C01823=1131.595,336.881,-80.038,-177.462,10.810,149.511
C01824=1131.592,337.129,-80.073,-177.459,10.813,149.510
C01825=1131.587,337.377,-80.107,-177.456,10.816,149.510
C01826=1131.583,337.624,-80.141,-177.452,10.818,149.510
C01827=1131.579,337.872,-80.176,-177.449,10.821,149.510
C01828=1131.576,338.119,-80.210,-177.446,10.823,149.510
C01829=1131.572,338.367,-80.244,-177.442,10.826,149.509
C01830=1131.568,338.614,-80.278,-177.439,10.828,149.509
C01831=1131.564,338.862,-80.313,-177.436,10.831,149.509
C01832=1131.560,339.109,-80.347,-177.433,10.833,149.509
C01833=1131.556,339.357,-80.382,-177.429,10.836,149.509
C01834=1131.552,339.605,-80.416,-177.426,10.838,149.508
C01835=1131.548,339.852,-80.450,-177.423,10.841,149.508
C01836=1131.544,340.100,-80.485,-177.421,10.843,149.508
C01837=1131.540,340.347,-80.519,-177.417,10.845,149.508
C01838=1131.536,340.595,-80.554,-177.414,10.847,149.508
C01839=1131.532,340.842,-80.588,-177.411,10.850,149.507
C01840=1131.528,341.091,-80.622,-177.407,10.852,149.507
C01841=1131.524,341.338,-80.657,-177.404,10.855,149.507
C01842=1131.520,341.586,-80.691,-177.401,10.858,149.507
C01843=1131.516,341.833,-80.726,-177.398,10.860,149.507
C01844=1131.512,342.081,-80.760,-177.394,10.863,149.506
C01845=1131.508,342.328,-80.795,-177.391,10.865,149.506
C01846=1131.504,342.576,-80.830,-177.388,10.867,149.506
C01847=1131.500,342.823,-80.864,-177.385,10.870,149.506
C01848=1131.496,343.071,-80.898,-177.382,10.873,149.506
C01849=1131.492,343.319,-80.933,-177.378,10.875,149.505
C01850=1131.488,343.566,-80.969,-177.375,10.878,149.505
C01851=1131.484,343.813,-81.002,-177.372,10.880,149.505
C01852=1131.480,344.061,-81.037,-177.368,10.883,149.505
C01853=1131.476,344.309,-81.072,-177.365,10.885,149.505
C01854=1131.473,344.556,-81.107,-177.362,10.888,149.504
C01855=1131.469,344.804,-81.141,-177.359,10.890,149.504
C01856=1131.464,345.051,-81.176,-177.355,10.893,149.504
C01857=1131.461,345.299,-81.211,-177.352,10.895,149.504
C01858=1131.457,345.546,-81.245,-177.349,10.898,149.503
C01859=1131.453,345.794,-81.280,-177.345,10.900,149.503
C01860=1131.449,346.042,-81.316,-177.343,10.903,149.503
C01861=1131.445,346.289,-81.350,-177.339,10.905,149.503
C01862=1131.441,346.537,-81.386,-177.336,10.908,149.503
C01863=1131.437,346.784,-81.420,-177.333,10.910,149.502
C01864=1131.433,347.032,-81.454,-177.329,10.913,149.502
C01865=1131.430,347.279,-81.490,-177.326,10.915,149.502
C01866=1131.425,347.527,-81.524,-177.323,10.918,149.502
C01867=1131.421,347.774,-81.560,-177.319,10.920,149.502
C01868=1131.419,347.987,-81.590,-177.317,10.922,149.501
C01869=1131.414,348.200,-81.619,-177.314,10.924,149.501
C01870=1131.411,348.414,-81.650,-177.311,10.927,149.501
C01871=1131.408,348.626,-81.680,-177.309,10.928,149.501
C01872=1131.405,348.839,-81.710,-177.305,10.931,149.501
C01873=1131.401,349.052,-81.741,-177.303,10.933,149.501
C01874=1131.398,349.265,-81.770,-177.300,10.935,149.500
C01875=1131.395,349.478,-81.801,-177.297,10.937,149.500
C01876=1131.391,349.726,-81.836,-177.294,10.939,149.500
C01877=1131.386,349.973,-81.871,-177.290,10.943,149.500
C01878=1131.383,350.220,-81.906,-177.287,10.945,149.499
C01879=1131.379,350.469,-81.941,-177.282,10.948,149.499
C01880=1131.375,350.716,-81.977,-177.279,10.950,149.499
C01881=1131.371,350.963,-82.012,-177.275,10.954,149.499
C01882=1131.367,351.211,-82.047,-177.272,10.956,149.498
C01883=1131.363,351.459,-82.082,-177.268,10.958,149.498
C01884=1131.359,351.705,-82.118,-177.264,10.961,149.498
C01885=1131.355,351.953,-82.152,-177.261,10.964,149.498
C01886=1131.351,352.201,-82.188,-177.257,10.966,149.497
C01887=1131.348,352.448,-82.224,-177.253,10.969,149.497
C01888=1131.343,352.695,-82.259,-177.250,10.972,149.497
C01889=1131.340,352.943,-82.294,-177.247,10.974,149.497
C01890=1131.336,353.191,-82.329,-177.242,10.977,149.496
C01891=1131.332,353.438,-82.365,-177.239,10.980,149.496
C01892=1131.328,353.686,-82.400,-177.236,10.982,149.496
C01893=1131.324,353.933,-82.435,-177.231,10.985,149.495
C01894=1131.321,354.180,-82.471,-177.228,10.987,149.495
C01895=1131.317,354.428,-82.506,-177.225,10.990,149.495
C01896=1131.313,354.675,-82.542,-177.221,10.992,149.495
C01897=1131.310,354.923,-82.578,-177.217,10.995,149.494
C01898=1131.305,355.169,-82.613,-177.214,10.998,149.494
C01899=1131.302,355.417,-82.648,-177.210,11.000,149.494
C01900=1131.297,355.665,-82.684,-177.207,11.002,149.493
C01901=1131.294,355.912,-82.720,-177.203,11.006,149.493
C01902=1131.290,356.160,-82.756,-177.199,11.008,149.493
C01903=1131.286,356.407,-82.791,-177.196,11.010,149.493
C01904=1131.282,356.654,-82.826,-177.192,11.013,149.492
C01905=1131.278,356.902,-82.862,-177.189,11.015,149.492
C01906=1131.274,357.149,-82.898,-177.185,11.018,149.492
C01907=1131.270,357.397,-82.933,-177.181,11.020,149.492
C01908=1131.267,357.644,-82.969,-177.178,11.023,149.491
C01909=1131.263,357.892,-83.005,-177.175,11.025,149.491
C01910=1131.259,358.139,-83.040,-177.171,11.028,149.491
C01911=1131.255,358.387,-83.077,-177.168,11.030,149.491
C01912=1131.251,358.633,-83.112,-177.164,11.032,149.490
C01913=1131.247,358.881,-83.148,-177.161,11.035,149.490
C01914=1131.244,359.128,-83.183,-177.158,11.037,149.490
C01915=1131.239,359.376,-83.219,-177.154,11.040,149.490
C01916=1131.236,359.623,-83.256,-177.150,11.043,149.489
C01917=1131.232,359.871,-83.291,-177.147,11.045,149.489
C01918=1131.228,360.118,-83.327,-177.143,11.047,149.489
C01919=1131.224,360.366,-83.363,-177.140,11.050,149.488
C01920=1131.221,360.613,-83.399,-177.137,11.052,149.488
C01921=1131.217,360.860,-83.435,-177.133,11.055,149.488
C01922=1131.213,361.108,-83.471,-177.130,11.057,149.488
C01923=1131.209,361.355,-83.507,-177.126,11.059,149.487
C01924=1131.206,361.568,-83.538,-177.124,11.061,149.487
C01925=1131.203,361.781,-83.569,-177.120,11.064,149.487
C01926=1131.199,361.993,-83.600,-177.118,11.066,149.487
C01927=1131.196,362.206,-83.630,-177.115,11.068,149.487
C01928=1131.193,362.419,-83.662,-177.112,11.070,149.486
C01929=1131.190,362.631,-83.693,-177.109,11.071,149.486
C01930=1131.186,362.845,-83.724,-177.106,11.074,149.486
C01931=1131.183,363.058,-83.755,-177.103,11.076,149.486
C01932=1131.179,363.305,-83.791,-177.100,11.078,149.485
C01933=1131.176,363.552,-83.827,-177.097,11.080,149.485
C01934=1131.171,363.800,-83.863,-177.093,11.083,149.485
C01935=1131.168,364.047,-83.900,-177.090,11.085,149.485
C01936=1131.163,364.295,-83.936,-177.086,11.088,149.484
C01937=1131.160,364.541,-83.972,-177.083,11.090,149.484
C01938=1131.156,364.789,-84.008,-177.080,11.093,149.484
C01939=1131.152,365.036,-84.044,-177.077,11.095,149.484
C01940=1131.148,365.283,-84.081,-177.074,11.097,149.484
C01941=1131.145,365.531,-84.117,-177.070,11.099,149.483
C01942=1131.141,365.778,-84.154,-177.067,11.101,149.483
C01943=1131.137,366.025,-84.189,-177.064,11.104,149.483
C01944=1131.133,366.273,-84.226,-177.060,11.106,149.483
C01945=1131.130,366.520,-84.263,-177.057,11.109,149.482
C01946=1131.126,366.768,-84.299,-177.054,11.111,149.482
C01947=1131.122,367.015,-84.335,-177.051,11.113,149.482
C01948=1131.118,367.262,-84.372,-177.048,11.115,149.482
C01949=1131.115,367.510,-84.408,-177.044,11.118,149.481
C01950=1131.110,367.757,-84.444,-177.041,11.120,149.481
C01951=1131.106,368.004,-84.481,-177.038,11.123,149.481
C01952=1131.103,368.251,-84.518,-177.035,11.124,149.481
C01953=1131.099,368.499,-84.554,-177.032,11.127,149.481
C01954=1131.095,368.746,-84.590,-177.029,11.129,149.480
C01955=1131.092,368.993,-84.627,-177.025,11.132,149.480
C01956=1131.088,369.241,-84.664,-177.023,11.134,149.480
C01957=1131.084,369.488,-84.700,-177.019,11.136,149.480
C01958=1131.080,369.735,-84.736,-177.016,11.139,149.479
C01959=1131.076,369.982,-84.773,-177.013,11.141,149.479
C01960=1131.072,370.229,-84.810,-177.010,11.143,149.479
C01961=1131.068,370.477,-84.846,-177.007,11.145,149.479
C01962=1131.066,370.724,-84.883,-177.003,11.148,149.479
C01963=1131.061,370.971,-84.920,-177.000,11.150,149.478
C01964=1131.057,371.219,-84.957,-176.997,11.152,149.478
C01965=1131.053,371.466,-84.994,-176.994,11.154,149.478
C01966=1131.050,371.713,-85.030,-176.991,11.157,149.478
C01967=1131.046,371.961,-85.066,-176.989,11.159,149.478
C01968=1131.042,372.208,-85.103,-176.985,11.161,149.477
C01969=1131.039,372.455,-85.139,-176.982,11.164,149.477
C01970=1131.035,372.702,-85.176,-176.979,11.166,149.477
C01971=1131.030,372.950,-85.213,-176.976,11.168,149.477
C01972=1131.027,373.198,-85.250,-176.973,11.170,149.477
C01973=1131.024,373.444,-85.287,-176.970,11.173,149.477
C01974=1131.020,373.691,-85.324,-176.967,11.175,149.476
C01975=1131.016,373.938,-85.361,-176.964,11.177,149.476
C01976=1131.012,374.185,-85.398,-176.961,11.179,149.476
C01977=1131.009,374.433,-85.435,-176.958,11.182,149.476
C01978=1131.005,374.680,-85.471,-176.955,11.184,149.476
C01979=1131.001,374.927,-85.508,-176.952,11.186,149.475
C01980=1130.997,375.140,-85.540,-176.950,11.188,149.475
C01981=1130.994,375.352,-85.572,-176.947,11.191,149.475
C01982=1130.991,375.565,-85.603,-176.944,11.193,149.475
C01983=1130.988,375.779,-85.636,-176.942,11.195,149.475
C01984=1130.985,375.991,-85.668,-176.939,11.196,149.475
C01985=1130.981,376.204,-85.700,-176.937,11.198,149.475
C01986=1130.978,376.416,-85.731,-176.935,11.200,149.474
C01987=1130.975,376.629,-85.763,-176.932,11.202,149.474
C01988=1130.971,376.876,-85.800,-176.929,11.205,149.474
C01989=1130.967,377.124,-85.838,-176.927,11.207,149.474
C01990=1130.963,377.371,-85.874,-176.923,11.209,149.474
C01991=1130.960,377.618,-85.911,-176.921,11.211,149.474
C01992=1130.956,377.864,-85.948,-176.918,11.214,149.474
C01993=1130.953,378.112,-85.985,-176.915,11.216,149.474
C01994=1130.948,378.359,-86.022,-176.912,11.218,149.473
C01995=1130.945,378.606,-86.060,-176.909,11.221,149.473
C01996=1130.941,378.854,-86.097,-176.907,11.223,149.473
C01997=1130.937,379.101,-86.134,-176.904,11.225,149.473
C01998=1130.933,379.348,-86.172,-176.901,11.227,149.473
C01999=1130.930,379.596,-86.209,-176.898,11.230,149.473
C02000=1130.926,379.843,-86.246,-176.896,11.232,149.473
C02001=1130.922,380.089,-86.283,-176.893,11.235,149.473
C02002=1130.918,380.337,-86.320,-176.890,11.236,149.473
C02003=1130.915,380.584,-86.358,-176.887,11.239,149.473
C02004=1130.911,380.831,-86.395,-176.885,11.241,149.473
C02005=1130.907,381.078,-86.433,-176.882,11.244,149.472
C02006=1130.903,381.325,-86.470,-176.880,11.246,149.472
C02007=1130.899,381.573,-86.506,-176.877,11.249,149.472
C02008=1130.896,381.820,-86.544,-176.874,11.251,149.472
C02009=1130.892,382.067,-86.581,-176.871,11.253,149.472
C02010=1130.889,382.314,-86.619,-176.869,11.255,149.472
C02011=1130.885,382.562,-86.656,-176.866,11.258,149.472
C02012=1130.881,382.808,-86.694,-176.864,11.260,149.472
C02013=1130.878,383.055,-86.732,-176.861,11.263,149.472
C02014=1130.874,383.303,-86.768,-176.859,11.265,149.472
C02015=1130.870,383.550,-86.806,-176.856,11.267,149.472
C02016=1130.866,383.797,-86.843,-176.855,11.268,149.472
C02017=1130.862,384.044,-86.881,-176.854,11.270,149.472
C02018=1130.858,384.292,-86.919,-176.853,11.272,149.472
C02019=1130.854,384.538,-86.956,-176.852,11.273,149.472
C02020=1130.851,384.786,-86.994,-176.850,11.275,149.472
C02021=1130.847,385.033,-87.031,-176.849,11.277,149.473
C02022=1130.844,385.280,-87.069,-176.847,11.279,149.473
C02023=1130.840,385.527,-87.106,-176.846,11.281,149.473
C02024=1130.836,385.774,-87.143,-176.845,11.282,149.473
C02025=1130.833,386.021,-87.181,-176.844,11.284,149.473
C02026=1130.829,386.268,-87.218,-176.843,11.286,149.473
C02027=1130.825,386.516,-87.257,-176.842,11.288,149.473
C02028=1130.821,386.762,-87.294,-176.841,11.289,149.474
C02029=1130.818,387.010,-87.332,-176.840,11.291,149.474
C02030=1130.814,387.257,-87.369,-176.838,11.293,149.474
C02031=1130.811,387.504,-87.407,-176.837,11.295,149.474
C02032=1130.807,387.751,-87.444,-176.836,11.297,149.474
C02033=1130.803,387.999,-87.482,-176.835,11.299,149.475
C02034=1130.799,388.246,-87.520,-176.834,11.301,149.475
C02035=1130.795,388.492,-87.558,-176.833,11.303,149.475
C02036=1130.793,388.705,-87.589,-176.832,11.304,149.475
C02037=1130.789,388.918,-87.622,-176.831,11.306,149.475
C02038=1130.786,389.130,-87.654,-176.830,11.308,149.476
C02039=1130.782,389.342,-87.687,-176.830,11.309,149.476
C02040=1130.780,389.555,-87.719,-176.829,11.311,149.476
C02041=1130.776,389.768,-87.751,-176.828,11.313,149.477
C02042=1130.773,389.981,-87.784,-176.827,11.315,149.477
C02043=1130.769,390.193,-87.816,-176.827,11.317,149.477
C02044=1130.766,390.440,-87.854,-176.826,11.319,149.477
C02045=1130.762,390.687,-87.892,-176.825,11.320,149.478
C02046=1130.759,390.935,-87.929,-176.824,11.322,149.478
C02047=1130.755,391.181,-87.967,-176.824,11.325,149.478
C02048=1130.751,391.429,-88.005,-176.822,11.327,149.479
C02049=1130.747,391.675,-88.043,-176.822,11.329,149.479
C02050=1130.744,391.923,-88.080,-176.821,11.331,149.479
C02051=1130.740,392.170,-88.118,-176.820,11.334,149.480
C02052=1130.737,392.417,-88.156,-176.819,11.335,149.480
C02053=1130.732,392.664,-88.194,-176.818,11.339,149.481
C02054=1130.729,392.911,-88.232,-176.817,11.340,149.481
C02055=1130.725,393.158,-88.269,-176.817,11.343,149.481
C02056=1130.722,393.406,-88.306,-176.817,11.345,149.482
C02057=1130.717,393.653,-88.345,-176.816,11.347,149.482
C02058=1130.714,393.900,-88.383,-176.815,11.350,149.483
C02059=1130.710,394.146,-88.420,-176.815,11.352,149.483
C02060=1130.707,394.394,-88.458,-176.814,11.355,149.484
C02061=1130.703,394.641,-88.496,-176.814,11.357,149.484
C02062=1130.699,394.888,-88.534,-176.813,11.359,149.485
C02063=1130.696,395.136,-88.571,-176.812,11.362,149.485
C02064=1130.692,395.382,-88.609,-176.812,11.364,149.486
C02065=1130.688,395.630,-88.648,-176.811,11.366,149.486
C02066=1130.684,395.876,-88.685,-176.811,11.369,149.487
C02067=1130.681,396.124,-88.723,-176.810,11.372,149.487
C02068=1130.677,396.371,-88.761,-176.810,11.374,149.488
C02069=1130.674,396.618,-88.799,-176.809,11.377,149.488
C02070=1130.670,396.864,-88.837,-176.809,11.379,149.489
C02071=1130.667,397.112,-88.875,-176.808,11.382,149.490
C02072=1130.662,397.359,-88.913,-176.808,11.385,149.490
C02073=1130.659,397.606,-88.951,-176.808,11.387,149.491
C02074=1130.655,397.853,-88.988,-176.807,11.391,149.491
C02075=1130.651,398.101,-89.026,-176.807,11.393,149.492
C02076=1130.647,398.347,-89.064,-176.807,11.396,149.493
C02077=1130.644,398.594,-89.102,-176.807,11.398,149.493
C02078=1130.640,398.842,-89.140,-176.806,11.402,149.494
C02079=1130.636,399.089,-89.178,-176.806,11.404,149.495
C02080=1130.633,399.336,-89.216,-176.806,11.407,149.495
C02081=1130.628,399.583,-89.254,-176.805,11.410,149.496
C02082=1130.625,399.830,-89.292,-176.805,11.413,149.497
C02083=1130.621,400.077,-89.329,-176.805,11.415,149.497
C02084=1130.618,400.324,-89.368,-176.805,11.419,149.498
C02085=1130.614,400.571,-89.406,-176.805,11.421,149.499
C02086=1130.611,400.818,-89.443,-176.804,11.425,149.499
C02087=1130.607,401.066,-89.482,-176.804,11.428,149.500
C02088=1130.603,401.312,-89.520,-176.805,11.430,149.501
C02089=1130.600,401.559,-89.557,-176.804,11.434,149.502
C02090=1130.595,401.806,-89.596,-176.804,11.437,149.503
C02091=1130.592,402.054,-89.634,-176.805,11.440,149.503
C02092=1130.589,402.265,-89.667,-176.804,11.443,149.504
C02093=1130.586,402.478,-89.700,-176.804,11.445,149.505
C02094=1130.582,402.691,-89.732,-176.804,11.448,149.506
C02095=1130.579,402.903,-89.765,-176.804,11.451,149.506
C02096=1130.577,403.116,-89.797,-176.804,11.454,149.507
C02097=1130.573,403.328,-89.830,-176.804,11.456,149.508
C02098=1130.570,403.540,-89.863,-176.805,11.459,149.509
C02099=1130.567,403.754,-89.896,-176.805,11.462,149.509
C02100=1130.562,404.000,-89.934,-176.804,11.465,149.510
C02101=1130.560,404.247,-89.972,-176.805,11.469,149.511
C02102=1130.556,404.494,-90.010,-176.805,11.472,149.512
C02103=1130.552,404.741,-90.048,-176.805,11.476,149.513
C02104=1130.549,404.988,-90.086,-176.805,11.479,149.514
C02105=1130.544,405.235,-90.125,-176.806,11.482,149.515
C02106=1130.541,405.483,-90.162,-176.805,11.486,149.516
C02107=1130.537,405.729,-90.200,-176.806,11.489,149.517
C02108=1130.533,405.977,-90.239,-176.806,11.493,149.518
C02109=1130.530,406.223,-90.277,-176.807,11.497,149.519
C02110=1130.526,406.470,-90.315,-176.807,11.501,149.520
C02111=1130.523,406.718,-90.353,-176.807,11.503,149.521
C02112=1130.519,406.964,-90.391,-176.808,11.508,149.522
C02113=1130.515,407.212,-90.429,-176.809,11.511,149.523
C02114=1130.512,407.459,-90.467,-176.809,11.515,149.524
C02115=1130.507,407.706,-90.506,-176.809,11.518,149.525
C02116=1130.504,407.953,-90.544,-176.809,11.522,149.526
C02117=1130.500,408.200,-90.583,-176.810,11.526,149.527
C02118=1130.497,408.447,-90.620,-176.811,11.530,149.528
C02119=1130.493,408.694,-90.658,-176.811,11.534,149.530
C02120=1130.490,408.942,-90.697,-176.812,11.537,149.531
C02121=1130.486,409.187,-90.735,-176.812,11.542,149.532
C02122=1130.482,409.435,-90.774,-176.813,11.546,149.533
C02123=1130.478,409.682,-90.811,-176.813,11.549,149.534
C02124=1130.474,409.929,-90.850,-176.814,11.553,149.535
C02125=1130.471,410.177,-90.888,-176.814,11.558,149.537
C02126=1130.467,410.423,-90.927,-176.815,11.561,149.538
C02127=1130.464,410.670,-90.965,-176.816,11.566,149.539
C02128=1130.460,410.918,-91.003,-176.816,11.570,149.540
C02129=1130.456,411.164,-91.041,-176.818,11.574,149.542
C02130=1130.452,411.411,-91.080,-176.818,11.578,149.543
C02131=1130.449,411.658,-91.118,-176.819,11.582,149.544
C02132=1130.446,411.905,-91.155,-176.819,11.587,149.546
C02133=1130.442,412.153,-91.194,-176.821,11.591,149.547
C02134=1130.439,412.399,-91.233,-176.821,11.595,149.548
C02135=1130.434,412.646,-91.271,-176.822,11.600,149.550
C02136=1130.431,412.893,-91.309,-176.823,11.604,149.551
C02137=1130.427,413.140,-91.348,-176.824,11.608,149.552
C02138=1130.424,413.387,-91.386,-176.825,11.613,149.554
C02139=1130.420,413.634,-91.424,-176.826,11.617,149.555
C02140=1130.416,413.882,-91.462,-176.827,11.622,149.556
C02141=1130.412,414.128,-91.501,-176.828,11.627,149.558
C02142=1130.409,414.375,-91.539,-176.829,11.631,149.559
C02143=1130.407,414.623,-91.578,-176.830,11.636,149.561
C02144=1130.404,414.870,-91.615,-176.831,11.640,149.562
C02145=1130.404,415.116,-91.653,-176.832,11.645,149.564
C02146=1130.403,415.364,-91.691,-176.833,11.650,149.565
C02147=1130.403,415.611,-91.729,-176.834,11.655,149.567
C02148=1130.403,415.823,-91.762,-176.835,11.658,149.568
C02149=1130.404,416.036,-91.794,-176.837,11.662,149.569
C02150=1130.406,416.248,-91.827,-176.838,11.667,149.571
C02151=1130.407,416.460,-91.859,-176.839,11.671,149.572
C02152=1130.409,416.673,-91.891,-176.840,11.675,149.574
C02153=1130.412,416.885,-91.923,-176.841,11.679,149.575
C02154=1130.415,417.097,-91.955,-176.843,11.683,149.576
C02155=1130.418,417.309,-91.987,-176.843,11.688,149.578
C02156=1130.000,417.309,-92.050,-176.836,11.692,149.577
C02157=1129.996,417.097,-92.018,-176.834,11.688,149.576
C02158=1129.992,416.884,-91.986,-176.834,11.683,149.574
C02159=1129.991,416.672,-91.954,-176.832,11.679,149.573
C02160=1129.988,416.460,-91.921,-176.832,11.675,149.572
C02161=1129.987,416.248,-91.889,-176.830,11.671,149.570
C02162=1129.985,416.036,-91.857,-176.829,11.667,149.569
C02163=1129.984,415.823,-91.824,-176.828,11.663,149.568
C02164=1129.984,415.610,-91.792,-176.828,11.658,149.566
C02165=1129.984,415.363,-91.754,-176.826,11.653,149.565
C02166=1129.985,415.116,-91.716,-176.825,11.650,149.563
C02167=1129.985,414.870,-91.678,-176.824,11.645,149.562
C02168=1129.987,414.623,-91.639,-176.823,11.640,149.560
C02169=1129.990,414.375,-91.602,-176.822,11.635,149.559
C02170=1129.993,414.129,-91.563,-176.821,11.631,149.557
C02171=1129.996,413.881,-91.525,-176.820,11.626,149.556
C02172=1130.000,413.634,-91.486,-176.819,11.621,149.554
C02173=1130.004,413.388,-91.448,-176.819,11.617,149.553
C02174=1130.008,413.140,-91.410,-176.818,11.612,149.552
C02175=1130.011,412.893,-91.371,-176.816,11.608,149.550
C02176=1130.015,412.647,-91.333,-176.816,11.604,149.549
C02177=1130.019,412.399,-91.294,-176.815,11.599,149.548
C02178=1130.022,412.152,-91.256,-176.814,11.594,149.546
C02179=1130.027,411.905,-91.218,-176.814,11.590,149.545
C02180=1130.029,411.658,-91.179,-176.813,11.587,149.544
C02181=1130.033,411.411,-91.141,-176.812,11.582,149.542
C02182=1130.037,411.164,-91.103,-176.811,11.578,149.541
C02183=1130.041,410.917,-91.064,-176.811,11.573,149.540
C02184=1130.044,410.670,-91.026,-176.810,11.569,149.539
C02185=1130.048,410.423,-90.988,-176.809,11.565,149.537
C02186=1130.052,410.176,-90.950,-176.809,11.561,149.536
C02187=1130.055,409.929,-90.911,-176.808,11.557,149.535
C02188=1130.059,409.682,-90.873,-176.807,11.553,149.534
C02189=1130.062,409.435,-90.835,-176.807,11.549,149.532
C02190=1130.066,409.187,-90.797,-176.807,11.545,149.531
C02191=1130.070,408.941,-90.759,-176.806,11.541,149.530
C02192=1130.074,408.694,-90.720,-176.805,11.537,149.529
C02193=1130.077,408.447,-90.682,-176.805,11.533,149.528
C02194=1130.081,408.200,-90.644,-176.805,11.529,149.527
C02195=1130.085,407.952,-90.606,-176.804,11.526,149.526
C02196=1130.089,407.706,-90.567,-176.804,11.522,149.525
C02197=1130.092,407.459,-90.529,-176.804,11.518,149.524
C02198=1130.096,407.211,-90.491,-176.803,11.514,149.522
C02199=1130.100,406.965,-90.453,-176.803,11.510,149.521
C02200=1130.103,406.717,-90.415,-176.802,11.507,149.520
C02201=1130.107,406.470,-90.376,-176.802,11.503,149.519
C02202=1130.110,406.224,-90.338,-176.802,11.499,149.518
C02203=1130.114,405.976,-90.300,-176.802,11.496,149.517
C02204=1130.118,405.730,-90.262,-176.801,11.492,149.516
C02205=1130.121,405.483,-90.224,-176.801,11.489,149.515
C02206=1130.125,405.235,-90.186,-176.801,11.485,149.514
C02207=1130.129,404.988,-90.148,-176.800,11.482,149.513
C02208=1130.133,404.741,-90.110,-176.801,11.478,149.512
C02209=1130.136,404.494,-90.071,-176.800,11.475,149.512
C02210=1130.140,404.247,-90.033,-176.800,11.471,149.511
C02211=1130.143,404.000,-89.995,-176.801,11.468,149.510
C02212=1130.147,403.753,-89.957,-176.800,11.465,149.509
C02213=1130.150,403.540,-89.924,-176.800,11.462,149.508
C02214=1130.154,403.328,-89.892,-176.800,11.459,149.507
C02215=1130.157,403.116,-89.859,-176.800,11.456,149.507
C02216=1130.160,402.903,-89.825,-176.800,11.453,149.506
C02217=1130.163,402.691,-89.793,-176.800,11.450,149.505
C02218=1130.167,402.479,-89.760,-176.800,11.448,149.504
C02219=1130.169,402.266,-89.727,-176.800,11.445,149.504
C02220=1130.172,402.054,-89.695,-176.800,11.442,149.503
C02221=1130.177,401.807,-89.657,-176.801,11.439,149.502
C02222=1130.180,401.559,-89.619,-176.800,11.436,149.501
C02223=1130.184,401.312,-89.581,-176.800,11.433,149.501
C02224=1130.188,401.065,-89.543,-176.801,11.430,149.500
C02225=1130.191,400.818,-89.505,-176.800,11.427,149.499
C02226=1130.195,400.571,-89.467,-176.801,11.424,149.498
C02227=1130.198,400.324,-89.429,-176.801,11.421,149.498
C02228=1130.202,400.077,-89.391,-176.801,11.417,149.497
C02229=1130.206,399.830,-89.353,-176.802,11.415,149.496
C02230=1130.209,399.582,-89.315,-176.802,11.412,149.496
C02231=1130.213,399.336,-89.277,-176.802,11.409,149.495
C02232=1130.217,399.088,-89.239,-176.802,11.406,149.494
C02233=1130.221,398.842,-89.201,-176.802,11.404,149.494
C02234=1130.224,398.594,-89.163,-176.803,11.400,149.493
C02235=1130.229,398.347,-89.125,-176.803,11.398,149.492
C02236=1130.232,398.100,-89.087,-176.804,11.394,149.492
C02237=1130.235,397.853,-89.049,-176.804,11.392,149.491
C02238=1130.239,397.606,-89.011,-176.804,11.390,149.490
C02239=1130.243,397.359,-88.973,-176.805,11.386,149.490
C02240=1130.246,397.112,-88.936,-176.805,11.384,149.489
C02241=1130.250,396.865,-88.897,-176.806,11.382,149.489
C02242=1130.254,396.618,-88.859,-176.806,11.379,149.488
C02243=1130.257,396.371,-88.822,-176.807,11.376,149.487
C02244=1130.261,396.124,-88.784,-176.807,11.374,149.487
C02245=1130.265,395.877,-88.745,-176.807,11.371,149.486
C02246=1130.269,395.630,-88.708,-176.808,11.368,149.486
C02247=1130.272,395.383,-88.670,-176.809,11.366,149.485
C02248=1130.277,395.136,-88.632,-176.809,11.364,149.485
C02249=1130.280,394.888,-88.595,-176.810,11.360,149.484
C02250=1130.283,394.641,-88.557,-176.811,11.358,149.484
C02251=1130.287,394.394,-88.519,-176.811,11.356,149.483
C02252=1130.291,394.147,-88.480,-176.811,11.354,149.483
C02253=1130.295,393.900,-88.443,-176.813,11.351,149.483
C02254=1130.298,393.653,-88.405,-176.813,11.349,149.482
C02255=1130.302,393.406,-88.367,-176.814,11.347,149.482
C02256=1130.306,393.158,-88.330,-176.814,11.344,149.481
C02257=1130.310,392.911,-88.292,-176.815,11.341,149.481
C02258=1130.313,392.664,-88.254,-176.816,11.339,149.480
C02259=1130.317,392.418,-88.216,-176.817,11.337,149.480
C02260=1130.321,392.170,-88.178,-176.818,11.335,149.480
C02261=1130.324,391.923,-88.140,-176.819,11.332,149.479
C02262=1130.328,391.676,-88.103,-176.820,11.330,149.479
C02263=1130.332,391.429,-88.066,-176.820,11.328,149.478
C02264=1130.335,391.182,-88.028,-176.821,11.326,149.478
C02265=1130.339,390.935,-87.989,-176.822,11.324,149.478
C02266=1130.343,390.688,-87.952,-176.823,11.322,149.478
C02267=1130.347,390.440,-87.915,-176.824,11.319,149.477
C02268=1130.350,390.193,-87.877,-176.825,11.318,149.477
C02269=1130.353,389.981,-87.844,-176.825,11.316,149.477
C02270=1130.357,389.768,-87.812,-176.826,11.314,149.476
C02271=1130.360,389.556,-87.780,-176.827,11.312,149.476
C02272=1130.362,389.343,-87.747,-176.828,11.311,149.476
C02273=1130.366,389.130,-87.715,-176.829,11.309,149.476
C02274=1130.370,388.918,-87.682,-176.829,11.307,149.475
C02275=1130.372,388.706,-87.650,-176.830,11.305,149.475
C02276=1130.375,388.493,-87.617,-176.832,11.304,149.475
C02277=1130.379,388.246,-87.580,-176.832,11.302,149.475
C02278=1130.383,387.999,-87.543,-176.833,11.300,149.474
C02279=1130.386,387.752,-87.505,-176.834,11.298,149.474
C02280=1130.391,387.505,-87.467,-176.836,11.296,149.474
C02281=1130.394,387.257,-87.429,-176.837,11.294,149.474
C02282=1130.398,387.011,-87.392,-176.838,11.292,149.474
C02283=1130.401,386.763,-87.354,-176.839,11.290,149.473
C02284=1130.405,386.516,-87.317,-176.840,11.289,149.473
C02285=1130.409,386.269,-87.279,-176.841,11.287,149.473
C02286=1130.412,386.022,-87.242,-176.843,11.285,149.473
C02287=1130.417,385.774,-87.204,-176.844,11.283,149.473
C02288=1130.420,385.527,-87.166,-176.845,11.281,149.473
C02289=1130.424,385.281,-87.129,-176.846,11.279,149.472
C02290=1130.428,385.033,-87.091,-176.848,11.278,149.472
C02291=1130.432,384.786,-87.054,-176.849,11.276,149.472
C02292=1130.435,384.539,-87.017,-176.850,11.275,149.472
C02293=1130.439,384.292,-86.979,-176.852,11.272,149.472
C02294=1130.442,384.045,-86.941,-176.853,11.270,149.472
C02295=1130.446,383.798,-86.904,-176.854,11.269,149.472
C02296=1130.450,383.551,-86.867,-176.855,11.267,149.472
C02297=1130.453,383.303,-86.829,-176.858,11.265,149.472
C02298=1130.458,383.056,-86.791,-176.860,11.263,149.472
C02299=1130.461,382.808,-86.754,-176.863,11.260,149.472
C02300=1130.465,382.562,-86.716,-176.865,11.258,149.472
C02301=1130.469,382.315,-86.679,-176.868,11.256,149.472
C02302=1130.472,382.067,-86.642,-176.871,11.254,149.472
C02303=1130.476,381.821,-86.604,-176.873,11.251,149.472
C02304=1130.480,381.573,-86.567,-176.876,11.249,149.472
C02305=1130.484,381.326,-86.530,-176.879,11.246,149.472
C02306=1130.488,381.079,-86.492,-176.881,11.245,149.472
C02307=1130.491,380.831,-86.455,-176.884,11.242,149.472
C02308=1130.495,380.585,-86.418,-176.886,11.240,149.472
C02309=1130.499,380.337,-86.381,-176.890,11.237,149.473
C02310=1130.502,380.090,-86.343,-176.892,11.235,149.473
C02311=1130.506,379.843,-86.306,-176.895,11.232,149.473
C02312=1130.510,379.596,-86.269,-176.898,11.231,149.473
C02313=1130.514,379.348,-86.231,-176.900,11.228,149.473
C02314=1130.518,379.101,-86.194,-176.903,11.226,149.473
C02315=1130.521,378.855,-86.157,-176.906,11.223,149.473
C02316=1130.525,378.607,-86.120,-176.908,11.221,149.473
C02317=1130.529,378.360,-86.083,-176.912,11.219,149.473
C02318=1130.533,378.112,-86.046,-176.915,11.216,149.473
C02319=1130.536,377.865,-86.008,-176.917,11.214,149.474
C02320=1130.540,377.618,-85.972,-176.920,11.212,149.474
C02321=1130.544,377.371,-85.935,-176.923,11.210,149.474
C02322=1130.547,377.124,-85.897,-176.926,11.207,149.474
C02323=1130.551,376.877,-85.860,-176.928,11.205,149.474
C02324=1130.555,376.629,-85.823,-176.931,11.203,149.474
C02325=1130.558,376.417,-85.792,-176.934,11.201,149.475
C02326=1130.562,376.204,-85.759,-176.936,11.199,149.475
C02327=1130.565,375.992,-85.728,-176.939,11.197,149.475
C02328=1130.569,375.779,-85.696,-176.941,11.195,149.475
C02329=1130.571,375.566,-85.664,-176.944,11.192,149.475
C02330=1130.574,375.353,-85.632,-176.947,11.191,149.475
C02331=1130.578,375.140,-85.601,-176.949,11.189,149.475
C02332=1130.581,374.928,-85.568,-176.952,11.187,149.475
C02333=1130.584,374.681,-85.532,-176.955,11.184,149.475
C02334=1130.588,374.434,-85.495,-176.957,11.182,149.476
C02335=1130.593,374.187,-85.458,-176.960,11.180,149.476
C02336=1130.596,373.939,-85.421,-176.963,11.178,149.476
C02337=1130.600,373.692,-85.384,-176.966,11.175,149.476
C02338=1130.603,373.445,-85.348,-176.969,11.173,149.476
C02339=1130.608,373.198,-85.311,-176.972,11.171,149.477
C02340=1130.611,372.950,-85.274,-176.975,11.169,149.477
C02341=1130.615,372.703,-85.237,-176.979,11.166,149.477
C02342=1130.619,372.456,-85.200,-176.981,11.164,149.477
C02343=1130.623,372.209,-85.164,-176.984,11.162,149.477
C02344=1130.627,371.961,-85.127,-176.988,11.159,149.478
C02345=1130.630,371.713,-85.089,-176.991,11.157,149.478
C02346=1130.634,371.467,-85.053,-176.993,11.155,149.478
C02347=1130.638,371.219,-85.016,-176.997,11.153,149.478
C02348=1130.642,370.972,-84.980,-177.000,11.150,149.478
C02349=1130.645,370.725,-84.943,-177.002,11.148,149.478
C02350=1130.649,370.478,-84.906,-177.006,11.146,149.479
C02351=1130.653,370.230,-84.869,-177.009,11.143,149.479
C02352=1130.656,369.983,-84.833,-177.012,11.141,149.479
C02353=1130.660,369.736,-84.797,-177.015,11.139,149.479
C02354=1130.665,369.488,-84.760,-177.018,11.137,149.480
C02355=1130.668,369.242,-84.724,-177.022,11.134,149.480
C02356=1130.672,368.994,-84.687,-177.025,11.132,149.480
C02357=1130.675,368.747,-84.651,-177.027,11.130,149.480
C02358=1130.679,368.499,-84.614,-177.031,11.127,149.480
C02359=1130.683,368.252,-84.577,-177.034,11.125,149.481
C02360=1130.687,368.005,-84.541,-177.037,11.122,149.481
C02361=1130.691,367.758,-84.504,-177.041,11.120,149.481
C02362=1130.694,367.510,-84.468,-177.043,11.118,149.481
C02363=1130.698,367.263,-84.432,-177.047,11.116,149.481
C02364=1130.703,367.016,-84.395,-177.050,11.113,149.482
C02365=1130.706,366.768,-84.359,-177.054,11.111,149.482
C02366=1130.710,366.521,-84.322,-177.057,11.109,149.482
C02367=1130.714,366.274,-84.286,-177.060,11.106,149.483
C02368=1130.718,366.026,-84.250,-177.063,11.105,149.483
C02369=1130.721,365.779,-84.213,-177.066,11.102,149.483
C02370=1130.725,365.532,-84.176,-177.070,11.100,149.483
C02371=1130.729,365.284,-84.141,-177.073,11.097,149.483
C02372=1130.733,365.037,-84.104,-177.076,11.095,149.484
C02373=1130.736,364.789,-84.069,-177.079,11.092,149.484
C02374=1130.740,364.542,-84.032,-177.083,11.090,149.484
C02375=1130.744,364.295,-83.996,-177.086,11.088,149.484
C02376=1130.748,364.048,-83.959,-177.090,11.085,149.485
C02377=1130.752,363.801,-83.923,-177.092,11.083,149.485
C02378=1130.755,363.553,-83.887,-177.096,11.081,149.485
C02379=1130.760,363.305,-83.851,-177.099,11.078,149.485
C02380=1130.763,363.058,-83.815,-177.103,11.076,149.486
C02381=1130.766,362.846,-83.784,-177.106,11.074,149.486
C02382=1130.769,362.633,-83.753,-177.108,11.072,149.486
C02383=1130.772,362.420,-83.722,-177.112,11.069,149.486
C02384=1130.775,362.207,-83.691,-177.114,11.068,149.486
C02385=1130.780,361.994,-83.660,-177.117,11.066,149.487
C02386=1130.783,361.782,-83.629,-177.120,11.064,149.487
C02387=1130.787,361.568,-83.598,-177.123,11.062,149.487
C02388=1130.790,361.356,-83.567,-177.126,11.059,149.487
C02389=1130.793,361.108,-83.531,-177.130,11.057,149.488
C02390=1130.797,360.861,-83.495,-177.133,11.054,149.488
C02391=1130.801,360.614,-83.459,-177.137,11.052,149.488
C02392=1130.805,360.366,-83.423,-177.140,11.050,149.488
C02393=1130.808,360.119,-83.387,-177.143,11.047,149.489
C02394=1130.812,359.871,-83.351,-177.147,11.045,149.489
C02395=1130.816,359.624,-83.315,-177.150,11.043,149.489
C02396=1130.820,359.376,-83.280,-177.154,11.040,149.490
C02397=1130.823,359.130,-83.243,-177.157,11.038,149.490
C02398=1130.827,358.882,-83.207,-177.160,11.035,149.490
C02399=1130.832,358.635,-83.172,-177.164,11.033,149.490
C02400=1130.835,358.387,-83.137,-177.167,11.031,149.491
C02401=1130.839,358.140,-83.101,-177.170,11.028,149.491
C02402=1130.843,357.893,-83.064,-177.174,11.025,149.491
C02403=1130.847,357.645,-83.029,-177.178,11.023,149.491
C02404=1130.851,357.398,-82.993,-177.181,11.020,149.492
C02405=1130.854,357.150,-82.958,-177.185,11.018,149.492
C02406=1130.858,356.903,-82.922,-177.188,11.016,149.492
C02407=1130.862,356.655,-82.886,-177.192,11.013,149.492
C02408=1130.866,356.408,-82.851,-177.195,11.011,149.493
C02409=1130.870,356.161,-82.815,-177.199,11.008,149.493
C02410=1130.874,355.913,-82.780,-177.203,11.006,149.493
C02411=1130.877,355.666,-82.744,-177.206,11.003,149.494
C02412=1130.881,355.418,-82.708,-177.209,11.001,149.494
C02413=1130.885,355.171,-82.673,-177.213,10.998,149.494
C02414=1130.890,354.923,-82.637,-177.217,10.995,149.494
C02415=1130.893,354.676,-82.602,-177.220,10.993,149.495
C02416=1130.897,354.428,-82.566,-177.224,10.990,149.495
C02417=1130.901,354.181,-82.531,-177.227,10.988,149.495
C02418=1130.904,353.933,-82.495,-177.231,10.985,149.495
C02419=1130.909,353.687,-82.460,-177.235,10.982,149.496
C02420=1130.912,353.439,-82.424,-177.238,10.980,149.496
C02421=1130.916,353.191,-82.389,-177.242,10.977,149.496
C02422=1130.920,352.944,-82.354,-177.245,10.975,149.496
C02423=1130.924,352.696,-82.318,-177.249,10.972,149.497
C02424=1130.928,352.449,-82.283,-177.253,10.969,149.497
C02425=1130.932,352.202,-82.248,-177.256,10.967,149.497
C02426=1130.936,351.954,-82.213,-177.260,10.964,149.497
C02427=1130.940,351.707,-82.178,-177.264,10.961,149.498
C02428=1130.943,351.459,-82.142,-177.267,10.959,149.498
C02429=1130.947,351.212,-82.106,-177.271,10.956,149.498
C02430=1130.951,350.964,-82.072,-177.275,10.953,149.498
C02431=1130.955,350.717,-82.036,-177.278,10.951,149.499
C02432=1130.959,350.469,-82.001,-177.282,10.948,149.499
C02433=1130.963,350.221,-81.966,-177.286,10.945,149.499
C02434=1130.967,349.975,-81.931,-177.289,10.943,149.500
C02435=1130.971,349.727,-81.895,-177.293,10.940,149.500
C02436=1130.975,349.479,-81.861,-177.297,10.938,149.500
C02437=1130.978,349.266,-81.831,-177.300,10.935,149.500
C02438=1130.981,349.053,-81.800,-177.302,10.933,149.500
C02439=1130.985,348.840,-81.770,-177.305,10.931,149.501
C02440=1130.988,348.628,-81.740,-177.308,10.929,149.501
C02441=1130.991,348.415,-81.710,-177.310,10.927,149.501
C02442=1130.995,348.201,-81.679,-177.314,10.925,149.501
C02443=1130.998,347.988,-81.650,-177.316,10.922,149.501
C02444=1131.002,347.775,-81.620,-177.319,10.920,149.502
C02445=1131.005,347.528,-81.584,-177.323,10.918,149.502
C02446=1131.010,347.280,-81.550,-177.326,10.915,149.502
C02447=1131.013,347.033,-81.515,-177.329,10.913,149.502
C02448=1131.017,346.786,-81.480,-177.332,10.910,149.502
C02449=1131.021,346.538,-81.445,-177.336,10.907,149.503
C02450=1131.025,346.290,-81.410,-177.338,10.906,149.503
C02451=1131.030,346.043,-81.375,-177.342,10.903,149.503
C02452=1131.032,345.795,-81.340,-177.345,10.901,149.503
C02453=1131.037,345.548,-81.306,-177.348,10.898,149.503
C02454=1131.041,345.300,-81.270,-177.351,10.896,149.504
C02455=1131.045,345.052,-81.236,-177.354,10.893,149.504
C02456=1131.049,344.805,-81.202,-177.358,10.891,149.504
C02457=1131.052,344.558,-81.166,-177.361,10.888,149.504
C02458=1131.057,344.310,-81.132,-177.364,10.886,149.504
C02459=1131.061,344.062,-81.097,-177.368,10.883,149.505
C02460=1131.065,343.815,-81.063,-177.371,10.881,149.505
C02461=1131.068,343.568,-81.027,-177.374,10.878,149.505
C02462=1131.073,343.320,-80.993,-177.377,10.876,149.505
C02463=1131.076,343.072,-80.959,-177.381,10.873,149.505
C02464=1131.080,342.824,-80.924,-177.384,10.871,149.506
C02465=1131.084,342.577,-80.889,-177.387,10.868,149.506
C02466=1131.088,342.329,-80.854,-177.390,10.866,149.506
C02467=1131.092,342.082,-80.820,-177.394,10.863,149.506
C02468=1131.096,341.834,-80.785,-177.397,10.861,149.506
C02469=1131.100,341.587,-80.751,-177.400,10.858,149.507
C02470=1131.104,341.339,-80.716,-177.403,10.856,149.507
C02471=1131.108,341.091,-80.682,-177.407,10.853,149.507
C02472=1131.112,340.844,-80.648,-177.410,10.851,149.507
C02473=1131.116,340.597,-80.613,-177.413,10.848,149.508
C02474=1131.120,340.350,-80.579,-177.416,10.845,149.508
C02475=1131.124,340.102,-80.544,-177.420,10.843,149.508
C02476=1131.128,339.854,-80.509,-177.423,10.841,149.508
C02477=1131.131,339.606,-80.475,-177.426,10.838,149.508
C02478=1131.136,339.359,-80.441,-177.429,10.836,149.509
C02479=1131.139,339.111,-80.406,-177.432,10.833,149.509
C02480=1131.144,338.864,-80.372,-177.436,10.830,149.509
C02481=1131.147,338.616,-80.338,-177.438,10.829,149.509
C02482=1131.152,338.368,-80.303,-177.442,10.826,149.509
C02483=1131.155,338.121,-80.269,-177.445,10.824,149.510
C02484=1131.160,337.873,-80.235,-177.448,10.821,149.510
C02485=1131.164,337.625,-80.201,-177.451,10.819,149.510
C02486=1131.168,337.377,-80.167,-177.455,10.816,149.510
C02487=1131.171,337.130,-80.133,-177.458,10.814,149.510
C02488=1131.175,336.882,-80.098,-177.461,10.811,149.511
C02489=1131.179,336.635,-80.064,-177.464,10.808,149.511
C02490=1131.184,336.388,-80.030,-177.467,10.806,149.511
C02491=1131.187,336.140,-79.995,-177.471,10.804,149.511
C02492=1131.191,335.892,-79.962,-177.474,10.801,149.511
C02493=1131.194,335.679,-79.932,-177.477,10.798,149.511
C02494=1131.198,335.466,-79.903,-177.480,10.797,149.512
C02495=1131.202,335.253,-79.874,-177.482,10.795,149.512
C02496=1131.204,335.039,-79.845,-177.485,10.792,149.512
C02497=1131.209,334.826,-79.815,-177.488,10.790,149.512
C02498=1131.211,334.613,-79.785,-177.491,10.788,149.512
C02499=1131.215,334.400,-79.756,-177.493,10.786,149.512
C02500=1131.218,334.187,-79.727,-177.496,10.784,149.513
C02501=1131.222,333.939,-79.693,-177.499,10.782,149.513
C02502=1131.226,333.692,-79.659,-177.502,10.779,149.513
C02503=1131.230,333.445,-79.626,-177.505,10.776,149.513
C02504=1131.235,333.196,-79.591,-177.509,10.774,149.514
C02505=1131.238,332.949,-79.558,-177.512,10.772,149.514
C02506=1131.242,332.702,-79.524,-177.515,10.769,149.514
C02507=1131.247,332.453,-79.490,-177.518,10.766,149.514
C02508=1131.250,332.206,-79.456,-177.522,10.764,149.514
C02509=1131.254,331.959,-79.422,-177.525,10.761,149.515
C02510=1131.258,331.710,-79.388,-177.528,10.759,149.515
C02511=1131.262,331.463,-79.354,-177.531,10.756,149.515
C02512=1131.266,331.215,-79.321,-177.535,10.754,149.515
C02513=1131.270,330.968,-79.287,-177.538,10.751,149.515
C02514=1131.274,330.719,-79.253,-177.541,10.748,149.515
C02515=1131.278,330.472,-79.219,-177.544,10.746,149.516
C02516=1131.283,330.224,-79.186,-177.547,10.744,149.516
C02517=1131.286,329.977,-79.152,-177.550,10.741,149.516
C02518=1131.290,329.729,-79.118,-177.554,10.738,149.516
C02519=1131.294,329.482,-79.084,-177.557,10.736,149.516
C02520=1131.299,329.234,-79.051,-177.560,10.733,149.517
C02521=1131.303,328.986,-79.017,-177.563,10.731,149.517
C02522=1131.306,328.738,-78.983,-177.567,10.728,149.517
C02523=1131.310,328.490,-78.950,-177.570,10.726,149.517
C02524=1131.314,328.243,-78.917,-177.572,10.724,149.517
C02525=1131.318,327.996,-78.883,-177.575,10.721,149.518
C02526=1131.322,327.747,-78.849,-177.579,10.719,149.518
C02527=1131.326,327.499,-78.816,-177.582,10.716,149.518
C02528=1131.330,327.252,-78.782,-177.585,10.714,149.518
C02529=1131.334,327.004,-78.749,-177.588,10.711,149.518
C02530=1131.339,326.757,-78.716,-177.592,10.709,149.519
C02531=1131.342,326.509,-78.682,-177.595,10.706,149.519
C02532=1131.346,326.261,-78.648,-177.598,10.704,149.519
C02533=1131.350,326.013,-78.615,-177.601,10.701,149.519
C02534=1131.354,325.766,-78.582,-177.604,10.698,149.519
C02535=1131.358,325.518,-78.548,-177.608,10.696,149.519
C02536=1131.362,325.271,-78.515,-177.611,10.693,149.520
C02537=1131.366,325.023,-78.482,-177.614,10.691,149.520
C02538=1131.370,324.775,-78.448,-177.617,10.688,149.520
C02539=1131.374,324.527,-78.415,-177.620,10.686,149.520
C02540=1131.378,324.279,-78.382,-177.624,10.683,149.521
C02541=1131.382,324.031,-78.349,-177.627,10.681,149.521
C02542=1131.386,323.784,-78.315,-177.630,10.678,149.521
C02543=1131.390,323.536,-78.282,-177.633,10.676,149.521
C02544=1131.394,323.289,-78.249,-177.636,10.673,149.521
C02545=1131.398,323.040,-78.215,-177.640,10.670,149.521
C02546=1131.402,322.793,-78.182,-177.643,10.668,149.522
C02547=1131.406,322.545,-78.149,-177.645,10.666,149.522
C02548=1131.410,322.297,-78.116,-177.649,10.664,149.522
C02549=1131.414,322.084,-78.087,-177.651,10.661,149.522
C02550=1131.418,321.871,-78.058,-177.654,10.659,149.522
C02551=1131.421,321.658,-78.031,-177.657,10.656,149.522
C02552=1131.424,321.444,-78.002,-177.660,10.655,149.523
C02553=1131.428,321.230,-77.974,-177.662,10.653,149.523
C02554=1131.431,321.018,-77.945,-177.665,10.650,149.523
C02555=1131.435,320.804,-77.916,-177.668,10.648,149.523
C02556=1131.438,320.591,-77.888,-177.671,10.645,149.523
C02557=1131.442,320.344,-77.855,-177.674,10.643,149.523
C02558=1131.446,320.096,-77.822,-177.677,10.641,149.524
C02559=1131.450,319.848,-77.789,-177.680,10.638,149.524
C02560=1131.455,319.600,-77.756,-177.683,10.636,149.524
C02561=1131.459,319.352,-77.723,-177.686,10.634,149.524
C02562=1131.463,319.105,-77.690,-177.689,10.631,149.524
C02563=1131.466,318.856,-77.657,-177.692,10.629,149.525
C02564=1131.470,318.609,-77.624,-177.696,10.626,149.525
C02565=1131.474,318.360,-77.591,-177.699,10.623,149.525
C02566=1131.478,318.113,-77.558,-177.702,10.621,149.525
C02567=1131.482,317.865,-77.526,-177.705,10.618,149.525
C02568=1131.486,317.617,-77.493,-177.708,10.616,149.526
C02569=1131.490,317.370,-77.459,-177.712,10.613,149.526
C02570=1131.494,317.121,-77.427,-177.715,10.610,149.526
C02571=1131.498,316.875,-77.395,-177.718,10.608,149.526
C02572=1131.503,316.627,-77.362,-177.721,10.606,149.526
C02573=1131.507,316.379,-77.329,-177.724,10.603,149.526
C02574=1131.510,316.131,-77.297,-177.727,10.600,149.527
C02575=1131.515,315.883,-77.263,-177.731,10.598,149.527
C02576=1131.519,315.635,-77.231,-177.734,10.595,149.527
C02577=1131.523,315.387,-77.198,-177.737,10.593,149.527
C02578=1131.527,315.139,-77.166,-177.740,10.590,149.527
C02579=1131.531,314.892,-77.133,-177.743,10.587,149.528
C02580=1131.534,314.644,-77.100,-177.746,10.586,149.528
C02581=1131.539,314.396,-77.068,-177.749,10.583,149.528
C02582=1131.543,314.148,-77.035,-177.752,10.581,149.528
C02583=1131.547,313.900,-77.003,-177.755,10.578,149.528
C02584=1131.551,313.652,-76.970,-177.758,10.575,149.529
C02585=1131.555,313.404,-76.937,-177.762,10.573,149.529
C02586=1131.559,313.157,-76.905,-177.765,10.570,149.529
C02587=1131.564,312.909,-76.873,-177.768,10.568,149.529
C02588=1131.567,312.661,-76.840,-177.771,10.565,149.529
C02589=1131.572,312.413,-76.808,-177.774,10.563,149.529
C02590=1131.576,312.165,-76.774,-177.778,10.560,149.530
C02591=1131.579,311.917,-76.743,-177.781,10.557,149.530
C02592=1131.584,311.669,-76.710,-177.784,10.555,149.530
C02593=1131.587,311.422,-76.678,-177.787,10.552,149.530
C02594=1131.592,311.174,-76.646,-177.790,10.550,149.530
C02595=1131.596,310.927,-76.613,-177.794,10.547,149.531
C02596=1131.600,310.678,-76.581,-177.796,10.544,149.531
C02597=1131.604,310.430,-76.549,-177.800,10.542,149.531
C02598=1131.608,310.182,-76.516,-177.802,10.540,149.531
C02599=1131.612,309.934,-76.484,-177.805,10.538,149.531
C02600=1131.617,309.687,-76.452,-177.808,10.535,149.531
C02601=1131.620,309.439,-76.419,-177.812,10.532,149.532
C02602=1131.625,309.191,-76.387,-177.815,10.530,149.532
C02603=1131.628,308.943,-76.355,-177.818,10.527,149.532
C02604=1131.633,308.695,-76.322,-177.821,10.525,149.532
C02605=1131.636,308.482,-76.295,-177.824,10.523,149.532
C02606=1131.640,308.269,-76.267,-177.826,10.520,149.532
C02607=1131.643,308.055,-76.239,-177.829,10.518,149.533
C02608=1131.647,307.842,-76.213,-177.832,10.516,149.533
C02609=1131.651,307.628,-76.184,-177.835,10.514,149.533
C02610=1131.654,307.415,-76.157,-177.837,10.512,149.533
C02611=1131.657,307.201,-76.129,-177.840,10.509,149.533
C02612=1131.661,306.988,-76.101,-177.843,10.508,149.534
C02613=1131.665,306.740,-76.069,-177.846,10.505,149.534
C02614=1131.669,306.492,-76.037,-177.849,10.502,149.534
C02615=1131.673,306.244,-76.005,-177.852,10.500,149.534
C02616=1131.677,305.996,-75.973,-177.855,10.497,149.534
C02617=1131.681,305.748,-75.941,-177.858,10.494,149.534
C02618=1131.685,305.501,-75.909,-177.862,10.492,149.535
C02619=1131.690,305.252,-75.877,-177.864,10.489,149.535
C02620=1131.694,305.004,-75.845,-177.868,10.487,149.535
C02621=1131.698,304.757,-75.814,-177.871,10.484,149.535
C02622=1131.702,304.509,-75.781,-177.874,10.482,149.535
C02623=1131.706,304.261,-75.749,-177.877,10.479,149.536
C02624=1131.710,304.013,-75.718,-177.880,10.477,149.536
C02625=1131.714,303.765,-75.686,-177.883,10.475,149.536
C02626=1131.719,303.517,-75.654,-177.886,10.472,149.536
C02627=1131.722,303.269,-75.622,-177.889,10.469,149.536
C02628=1131.727,303.021,-75.590,-177.892,10.467,149.536
C02629=1131.731,302.773,-75.558,-177.896,10.464,149.537
C02630=1131.735,302.525,-75.526,-177.898,10.461,149.537
C02631=1131.739,302.277,-75.495,-177.902,10.459,149.537
C02632=1131.743,302.029,-75.463,-177.905,10.456,149.537
C02633=1131.747,301.782,-75.432,-177.908,10.454,149.537
C02634=1131.752,301.533,-75.400,-177.911,10.451,149.538
C02635=1131.755,301.285,-75.368,-177.914,10.449,149.538
C02636=1131.760,301.038,-75.336,-177.918,10.446,149.538
C02637=1131.764,300.789,-75.305,-177.921,10.443,149.538
C02638=1131.768,300.542,-75.274,-177.924,10.441,149.538
C02639=1131.772,300.294,-75.242,-177.926,10.439,149.538
C02640=1131.776,300.046,-75.209,-177.930,10.437,149.539
C02641=1131.781,299.798,-75.179,-177.933,10.434,149.539
C02642=1131.785,299.550,-75.147,-177.936,10.431,149.539
C02643=1131.789,299.302,-75.115,-177.939,10.429,149.539
C02644=1131.793,299.054,-75.084,-177.942,10.426,149.539
C02645=1131.797,298.806,-75.052,-177.945,10.423,149.539
C02646=1131.801,298.558,-75.021,-177.948,10.421,149.540
C02647=1131.805,298.310,-74.990,-177.951,10.418,149.540
C02648=1131.809,298.062,-74.958,-177.955,10.416,149.540
C02649=1131.813,297.814,-74.926,-177.958,10.413,149.540
C02650=1131.818,297.566,-74.896,-177.961,10.411,149.540
C02651=1131.822,297.318,-74.863,-177.964,10.408,149.541
C02652=1131.826,297.069,-74.832,-177.967,10.405,149.541
C02653=1131.830,296.822,-74.801,-177.970,10.403,149.541
C02654=1131.834,296.574,-74.769,-177.973,10.401,149.541
C02655=1131.839,296.326,-74.738,-177.976,10.398,149.541
C02656=1131.842,296.078,-74.706,-177.979,10.396,149.542
C02657=1131.847,295.830,-74.675,-177.982,10.393,149.542
C02658=1131.850,295.582,-74.644,-177.985,10.391,149.542
C02659=1131.855,295.334,-74.613,-177.988,10.388,149.542
C02660=1131.858,295.086,-74.581,-177.992,10.385,149.542
C02661=1131.862,294.873,-74.555,-177.994,10.384,149.542
C02662=1131.866,294.659,-74.527,-177.997,10.381,149.542
C02663=1131.870,294.445,-74.501,-178.000,10.379,149.543
C02664=1131.873,294.231,-74.474,-178.002,10.377,149.543
C02665=1131.877,294.018,-74.447,-178.005,10.374,149.543
C02666=1131.881,293.804,-74.420,-178.007,10.372,149.543
C02667=1131.884,293.591,-74.394,-178.010,10.370,149.543
C02668=1131.888,293.377,-74.367,-178.013,10.368,149.543
C02669=1131.892,293.129,-74.335,-178.016,10.365,149.544
C02670=1131.896,292.882,-74.305,-178.019,10.363,149.544
C02671=1131.900,292.633,-74.274,-178.022,10.360,149.544
C02672=1131.904,292.386,-74.242,-178.025,10.358,149.544
C02673=1131.908,292.137,-74.211,-178.028,10.355,149.544
C02674=1131.912,291.889,-74.181,-178.031,10.353,149.545
C02675=1131.916,291.641,-74.149,-178.034,10.350,149.545
C02676=1131.920,291.393,-74.119,-178.037,10.348,149.545
C02677=1131.925,291.146,-74.088,-178.040,10.345,149.545
C02678=1131.929,290.897,-74.057,-178.044,10.343,149.545
C02679=1131.933,290.649,-74.026,-178.046,10.340,149.545
C02680=1131.937,290.401,-73.994,-178.050,10.338,149.546
C02681=1131.941,290.153,-73.964,-178.053,10.335,149.546
C02682=1131.946,289.905,-73.933,-178.056,10.332,149.546
C02683=1131.950,289.657,-73.902,-178.059,10.330,149.546
C02684=1131.954,289.409,-73.871,-178.062,10.327,149.546
C02685=1131.957,289.160,-73.841,-178.065,10.324,149.546
C02686=1131.962,288.913,-73.809,-178.068,10.322,149.547
C02687=1131.966,288.665,-73.778,-178.071,10.320,149.547
C02688=1131.970,288.416,-73.747,-178.074,10.317,149.547
C02689=1131.974,288.169,-73.717,-178.077,10.315,149.547
C02690=1131.979,287.921,-73.686,-178.080,10.312,149.547
C02691=1131.983,287.672,-73.655,-178.083,10.310,149.548
C02692=1131.987,287.424,-73.625,-178.086,10.307,149.548
C02693=1131.991,287.176,-73.594,-178.090,10.305,149.548
C02694=1131.995,286.928,-73.563,-178.093,10.302,149.548
C02695=1131.999,286.680,-73.533,-178.096,10.299,149.548
C02696=1132.004,286.432,-73.502,-178.099,10.297,149.548
C02697=1132.008,286.184,-73.471,-178.101,10.295,149.549
C02698=1132.012,285.936,-73.441,-178.105,10.292,149.549
C02699=1132.016,285.688,-73.410,-178.108,10.289,149.549
C02700=1132.021,285.440,-73.379,-178.111,10.287,149.549
C02701=1132.024,285.192,-73.349,-178.114,10.284,149.549
C02702=1132.029,284.944,-73.318,-178.117,10.282,149.550
C02703=1132.033,284.695,-73.289,-178.120,10.279,149.550
C02704=1132.038,284.447,-73.258,-178.123,10.276,149.550
C02705=1132.041,284.199,-73.227,-178.126,10.274,149.550
C02706=1132.046,283.951,-73.197,-178.129,10.271,149.550
C02707=1132.050,283.703,-73.166,-178.133,10.269,149.550
C02708=1132.054,283.456,-73.136,-178.135,10.267,149.551
C02709=1132.058,283.206,-73.105,-178.138,10.264,149.551
C02710=1132.062,282.959,-73.075,-178.141,10.262,149.551
C02711=1132.067,282.711,-73.044,-178.144,10.259,149.551
C02712=1132.071,282.463,-73.014,-178.148,10.256,149.551
C02713=1132.075,282.214,-72.984,-178.150,10.254,149.551
C02714=1132.079,281.966,-72.954,-178.154,10.251,149.552
C02715=1132.083,281.718,-72.923,-178.157,10.248,149.552
C02716=1132.087,281.470,-72.893,-178.160,10.246,149.552
C02717=1132.091,281.256,-72.866,-178.163,10.243,149.552
C02718=1132.095,281.042,-72.841,-178.166,10.241,149.552
C02719=1132.098,280.829,-72.814,-178.169,10.239,149.553
C02720=1132.102,280.615,-72.789,-178.172,10.236,149.553
C02721=1132.106,280.401,-72.762,-178.175,10.234,149.553
C02722=1132.109,280.188,-72.737,-178.178,10.231,149.553
C02723=1132.113,279.973,-72.710,-178.181,10.229,149.553
C02724=1132.116,279.761,-72.685,-178.185,10.226,149.554
C02725=1132.121,279.512,-72.655,-178.188,10.224,149.554
C02726=1132.125,279.264,-72.624,-178.192,10.220,149.554
C02727=1132.129,279.015,-72.594,-178.195,10.218,149.554
C02728=1132.133,278.767,-72.564,-178.198,10.214,149.554
C02729=1132.137,278.519,-72.534,-178.202,10.212,149.555
C02730=1132.142,278.271,-72.504,-178.205,10.209,149.555
C02731=1132.146,278.023,-72.474,-178.209,10.206,149.555
C02732=1132.150,277.775,-72.444,-178.212,10.203,149.555
C02733=1132.155,277.527,-72.414,-178.215,10.201,149.555
C02734=1132.159,277.279,-72.384,-178.219,10.197,149.556
C02735=1132.163,277.031,-72.354,-178.222,10.195,149.556
C02736=1132.166,276.782,-72.324,-178.225,10.192,149.556
C02737=1132.171,276.534,-72.294,-178.228,10.190,149.556
C02738=1132.175,276.286,-72.264,-178.232,10.186,149.556
C02739=1132.179,276.038,-72.234,-178.235,10.184,149.557
C02740=1132.184,275.790,-72.205,-178.238,10.181,149.557
C02741=1132.188,275.541,-72.175,-178.241,10.178,149.557
C02742=1132.192,275.293,-72.144,-178.244,10.176,149.557
C02743=1132.196,275.045,-72.115,-178.247,10.173,149.557
C02744=1132.201,274.797,-72.086,-178.251,10.169,149.557
C02745=1132.205,274.549,-72.055,-178.254,10.167,149.557
C02746=1132.209,274.301,-72.025,-178.257,10.164,149.558
C02747=1132.214,274.052,-71.996,-178.260,10.161,149.558
C02748=1132.218,273.804,-71.966,-178.263,10.159,149.558
C02749=1132.222,273.556,-71.937,-178.266,10.156,149.558
C02750=1132.226,273.308,-71.907,-178.269,10.154,149.558
C02751=1132.230,273.060,-71.877,-178.272,10.151,149.558
C02752=1132.235,272.811,-71.847,-178.275,10.148,149.558
C02753=1132.239,272.563,-71.818,-178.278,10.145,149.558
C02754=1132.243,272.315,-71.788,-178.281,10.142,149.559
C02755=1132.248,272.067,-71.759,-178.284,10.140,149.559
C02756=1132.251,271.819,-71.729,-178.286,10.138,149.559
C02757=1132.256,271.571,-71.699,-178.290,10.135,149.559
C02758=1132.260,271.322,-71.670,-178.293,10.133,149.559
C02759=1132.264,271.074,-71.640,-178.296,10.130,149.559
C02760=1132.268,270.826,-71.611,-178.298,10.127,149.559
C02761=1132.272,270.578,-71.581,-178.301,10.124,149.560
C02762=1132.276,270.329,-71.552,-178.304,10.122,149.560
C02763=1132.281,270.081,-71.523,-178.307,10.120,149.560
C02764=1132.286,269.832,-71.493,-178.310,10.117,149.560
C02765=1132.290,269.584,-71.463,-178.312,10.115,149.560
C02766=1132.295,269.337,-71.434,-178.315,10.112,149.560
C02767=1132.299,269.088,-71.405,-178.317,10.109,149.560
C02768=1132.303,268.840,-71.375,-178.320,10.107,149.560
C02769=1132.307,268.592,-71.346,-178.323,10.104,149.560
C02770=1132.311,268.344,-71.316,-178.326,10.101,149.560
C02771=1132.315,268.095,-71.287,-178.328,10.099,149.560
C02772=1132.320,267.847,-71.257,-178.331,10.097,149.561
C02773=1132.324,267.633,-71.233,-178.333,10.095,149.561
C02774=1132.327,267.420,-71.208,-178.335,10.092,149.561
C02775=1132.330,267.205,-71.182,-178.337,10.090,149.561
C02776=1132.335,266.991,-71.157,-178.340,10.088,149.561
C02777=1132.338,266.778,-71.132,-178.342,10.086,149.561
C02778=1132.342,266.564,-71.107,-178.344,10.084,149.561
C02779=1132.345,266.350,-71.081,-178.346,10.082,149.561
C02780=1132.349,266.136,-71.057,-178.348,10.080,149.561
C02781=1132.353,265.888,-71.027,-178.351,10.078,149.561
C02782=1132.357,265.640,-70.998,-178.353,10.076,149.561
C02783=1132.361,265.391,-70.968,-178.356,10.073,149.561
C02784=1132.366,265.143,-70.940,-178.358,10.071,149.561
C02785=1132.370,264.895,-70.910,-178.360,10.069,149.562
C02786=1132.375,264.647,-70.881,-178.363,10.067,149.562
C02787=1132.379,264.398,-70.852,-178.365,10.064,149.562
C02788=1132.383,264.149,-70.823,-178.369,10.061,149.562
C02789=1132.387,263.902,-70.794,-178.373,10.058,149.562
C02790=1132.392,263.654,-70.765,-178.377,10.055,149.563
C02791=1132.396,263.405,-70.736,-178.381,10.051,149.563
C02792=1132.400,263.157,-70.707,-178.385,10.048,149.563
C02793=1132.404,262.908,-70.677,-178.389,10.045,149.563
C02794=1132.409,262.661,-70.649,-178.393,10.042,149.564
C02795=1132.413,262.412,-70.620,-178.397,10.039,149.564
C02796=1132.417,262.164,-70.591,-178.401,10.035,149.564
C02797=1132.422,261.915,-70.562,-178.405,10.032,149.564
C02798=1132.426,261.668,-70.533,-178.407,10.029,149.564
C02799=1132.430,261.419,-70.505,-178.411,10.026,149.565
C02800=1132.434,261.171,-70.475,-178.415,10.023,149.565
C02801=1132.439,260.922,-70.446,-178.419,10.019,149.565
C02802=1132.443,260.675,-70.418,-178.422,10.017,149.565
C02803=1132.447,260.426,-70.389,-178.426,10.013,149.565
C02804=1132.451,260.177,-70.360,-178.429,10.011,149.566
C02805=1132.456,259.930,-70.332,-178.432,10.007,149.566
C02806=1132.460,259.681,-70.302,-178.436,10.004,149.566
C02807=1132.465,259.432,-70.274,-178.439,10.001,149.566
C02808=1132.468,259.184,-70.246,-178.443,9.998,149.566
C02809=1132.473,258.936,-70.216,-178.446,9.995,149.566
C02810=1132.478,258.687,-70.188,-178.449,9.992,149.566
C02811=1132.481,258.439,-70.160,-178.453,9.989,149.567
C02812=1132.486,258.191,-70.130,-178.456,9.986,149.567
C02813=1132.490,257.943,-70.102,-178.459,9.983,149.567
C02814=1132.494,257.694,-70.074,-178.462,9.980,149.567
C02815=1132.498,257.447,-70.045,-178.465,9.977,149.567
C02816=1132.503,257.198,-70.016,-178.468,9.974,149.567
C02817=1132.508,256.949,-69.988,-178.471,9.972,149.567
C02818=1132.512,256.701,-69.960,-178.474,9.969,149.567
C02819=1132.516,256.453,-69.930,-178.477,9.966,149.567
C02820=1132.520,256.205,-69.903,-178.480,9.963,149.567
C02821=1132.525,255.956,-69.874,-178.483,9.960,149.568
C02822=1132.528,255.707,-69.846,-178.482,9.960,149.567
C02823=1132.534,255.459,-69.817,-178.481,9.959,149.567
C02824=1132.537,255.211,-69.789,-178.480,9.958,149.566
C02825=1132.542,254.963,-69.760,-178.480,9.958,149.566
C02826=1132.546,254.714,-69.732,-178.479,9.957,149.566
C02827=1132.550,254.465,-69.703,-178.479,9.956,149.566
C02828=1132.555,254.218,-69.676,-178.480,9.955,149.565
C02829=1132.558,254.004,-69.650,-178.480,9.954,149.565
C02830=1132.562,253.790,-69.626,-178.481,9.952,149.565
C02831=1132.566,253.576,-69.601,-178.482,9.952,149.565
C02832=1132.570,253.362,-69.577,-178.483,9.950,149.565
C02833=1132.574,253.148,-69.552,-178.484,9.949,149.565
C02834=1132.577,252.933,-69.528,-178.485,9.947,149.565
C02835=1132.580,252.719,-69.504,-178.488,9.945,149.565
C02836=1132.584,252.505,-69.479,-178.490,9.943,149.565
C02837=1132.589,252.257,-69.451,-178.492,9.941,149.565
C02838=1132.593,252.009,-69.422,-178.495,9.938,149.566
C02839=1132.598,251.761,-69.394,-178.499,9.936,149.566
C02840=1132.601,251.513,-69.366,-178.502,9.933,149.566
C02841=1132.606,251.264,-69.337,-178.506,9.930,149.566
C02842=1132.610,251.016,-69.309,-178.510,9.927,149.567
C02843=1132.614,250.767,-69.281,-178.514,9.924,149.567
C02844=1132.619,250.519,-69.253,-178.519,9.920,149.567
C02845=1132.623,250.270,-69.224,-178.524,9.916,149.568
C02846=1132.627,250.023,-69.197,-178.529,9.913,149.568
C02847=1132.632,249.774,-69.168,-178.534,9.909,149.569
C02848=1132.636,249.526,-69.140,-178.540,9.904,149.569
C02849=1132.640,249.277,-69.111,-178.546,9.900,149.570
C02850=1132.645,249.029,-69.084,-178.552,9.895,149.570
C02851=1132.649,248.780,-69.056,-178.559,9.890,149.571
C02852=1132.653,248.532,-69.028,-178.566,9.885,149.571
C02853=1132.658,248.283,-69.000,-178.573,9.880,149.572
C02854=1132.662,248.035,-68.972,-178.580,9.874,149.573
C02855=1132.666,247.787,-68.944,-178.588,9.868,149.573
C02856=1132.670,247.538,-68.917,-178.596,9.862,149.574
C02857=1132.675,247.290,-68.889,-178.600,9.858,149.574
C02858=1132.679,247.041,-68.860,-178.601,9.856,149.574
C02859=1132.684,246.793,-68.833,-178.602,9.854,149.574
C02860=1132.688,246.545,-68.805,-178.603,9.852,149.573
C02861=1132.692,246.296,-68.778,-178.605,9.850,149.573
C02862=1132.697,246.048,-68.750,-178.606,9.848,149.573
C02863=1132.700,245.799,-68.722,-178.606,9.846,149.573
C02864=1132.706,245.551,-68.694,-178.608,9.844,149.573
C02865=1132.710,245.303,-68.667,-178.609,9.842,149.573
C02866=1132.714,245.054,-68.638,-178.611,9.840,149.573
C02867=1132.719,244.806,-68.611,-178.612,9.838,149.572
C02868=1132.723,244.558,-68.584,-178.613,9.836,149.572
C02869=1132.727,244.309,-68.556,-178.615,9.834,149.572
C02870=1132.731,244.061,-68.528,-178.617,9.831,149.572
C02871=1132.736,243.812,-68.501,-178.618,9.830,149.572
C02872=1132.740,243.564,-68.473,-178.620,9.827,149.572
C02873=1132.744,243.315,-68.446,-178.622,9.825,149.572
C02874=1132.750,243.067,-68.418,-178.623,9.823,149.572
C02875=1132.753,242.818,-68.390,-178.625,9.821,149.572
C02876=1132.758,242.570,-68.362,-178.627,9.819,149.572
C02877=1132.762,242.322,-68.335,-178.629,9.816,149.572
C02878=1132.766,242.073,-68.307,-178.630,9.814,149.571
C02879=1132.771,241.825,-68.279,-178.632,9.813,149.571
C02880=1132.775,241.576,-68.252,-178.634,9.810,149.571
C02881=1132.779,241.327,-68.225,-178.635,9.808,149.571
C02882=1132.784,241.079,-68.197,-178.638,9.806,149.571
C02883=1132.788,240.831,-68.170,-178.640,9.803,149.571
C02884=1132.792,240.582,-68.142,-178.642,9.800,149.571
C02885=1132.796,240.369,-68.119,-178.644,9.799,149.572
C02886=1132.800,240.155,-68.095,-178.646,9.797,149.571
C02887=1132.804,239.940,-68.072,-178.648,9.795,149.571
C02888=1132.808,239.725,-68.048,-178.650,9.793,149.572
C02889=1132.811,239.512,-68.024,-178.652,9.790,149.571
C02890=1132.815,239.297,-68.000,-178.654,9.788,149.572
C02891=1132.819,239.084,-67.977,-178.656,9.786,149.572
C02892=1132.823,238.869,-67.953,-178.658,9.784,149.572
C02893=1132.828,238.621,-67.926,-178.660,9.782,149.572
C02894=1132.831,238.372,-67.898,-178.663,9.779,149.572
C02895=1132.835,238.124,-67.871,-178.666,9.777,149.572
C02896=1132.840,237.876,-67.844,-178.668,9.774,149.572
C02897=1132.844,237.628,-67.816,-178.670,9.772,149.572
C02898=1132.848,237.379,-67.789,-178.673,9.769,149.572
C02899=1132.853,237.130,-67.762,-178.676,9.766,149.572
C02900=1132.858,236.882,-67.735,-178.679,9.764,149.572
C02901=1132.862,236.634,-67.707,-178.681,9.761,149.572
C02902=1132.866,236.384,-67.680,-178.684,9.759,149.572
C02903=1132.871,236.136,-67.653,-178.687,9.756,149.573
C02904=1132.875,235.887,-67.626,-178.690,9.753,149.573
C02905=1132.879,235.640,-67.598,-178.693,9.750,149.573
C02906=1132.884,235.391,-67.571,-178.696,9.748,149.573
C02907=1132.888,235.142,-67.544,-178.699,9.745,149.573
C02908=1132.892,234.894,-67.517,-178.702,9.741,149.573
C02909=1132.897,234.645,-67.490,-178.705,9.739,149.573
C02910=1132.902,234.397,-67.463,-178.709,9.736,149.574
C02911=1132.906,234.149,-67.436,-178.712,9.733,149.574
C02912=1132.910,233.899,-67.409,-178.715,9.730,149.574
C02913=1132.914,233.652,-67.381,-178.718,9.727,149.574
C02914=1132.919,233.403,-67.354,-178.722,9.724,149.574
C02915=1132.923,233.155,-67.328,-178.725,9.721,149.574
C02916=1132.927,232.906,-67.300,-178.729,9.718,149.575
C02917=1132.932,232.658,-67.273,-178.732,9.715,149.575
C02918=1132.936,232.409,-67.246,-178.735,9.711,149.575
C02919=1132.940,232.160,-67.220,-178.739,9.708,149.575
C02920=1132.944,231.912,-67.192,-178.742,9.706,149.575
C02921=1132.949,231.663,-67.165,-178.746,9.702,149.575
C02922=1132.954,231.414,-67.139,-178.749,9.699,149.575
C02923=1132.958,231.166,-67.113,-178.753,9.695,149.576
C02924=1132.963,230.918,-67.086,-178.757,9.692,149.576
C02925=1132.967,230.669,-67.058,-178.761,9.688,149.576
C02926=1132.971,230.421,-67.032,-178.764,9.685,149.576
C02927=1132.976,230.172,-67.005,-178.768,9.682,149.576
C02928=1132.980,229.924,-66.978,-178.772,9.677,149.577
C02929=1132.985,229.675,-66.952,-178.776,9.674,149.577
C02930=1132.989,229.427,-66.925,-178.780,9.671,149.577
C02931=1132.993,229.179,-66.899,-178.784,9.667,149.577
C02932=1132.998,228.930,-66.872,-178.788,9.663,149.577
C02933=1133.002,228.682,-66.845,-178.792,9.660,149.578
C02934=1133.007,228.433,-66.819,-178.795,9.656,149.578
C02935=1133.012,228.184,-66.792,-178.799,9.653,149.578
C02936=1133.015,227.936,-66.765,-178.802,9.649,149.578
C02937=1133.020,227.687,-66.739,-178.806,9.646,149.578
C02938=1133.024,227.439,-66.712,-178.810,9.642,149.578
C02939=1133.029,227.190,-66.685,-178.813,9.639,149.578
C02940=1133.033,226.941,-66.660,-178.817,9.635,149.578
C02941=1133.037,226.727,-66.636,-178.820,9.632,149.578
C02942=1133.041,226.513,-66.614,-178.823,9.629,149.579
C02943=1133.044,226.298,-66.591,-178.826,9.626,149.579
C02944=1133.048,226.084,-66.568,-178.829,9.623,149.579
C02945=1133.052,225.870,-66.545,-178.832,9.620,149.579
C02946=1133.056,225.655,-66.523,-178.834,9.617,149.579
C02947=1133.060,225.442,-66.500,-178.838,9.614,149.579
C02948=1133.063,225.227,-66.478,-178.841,9.611,149.579
C02949=1133.067,224.979,-66.451,-178.843,9.608,149.579
C02950=1133.072,224.730,-66.425,-178.847,9.604,149.579
C02951=1133.077,224.482,-66.399,-178.850,9.600,149.579
C02952=1133.081,224.233,-66.373,-178.853,9.598,149.579
C02953=1133.086,223.985,-66.346,-178.856,9.594,149.579
C02954=1133.090,223.736,-66.320,-178.860,9.590,149.579
C02955=1133.095,223.487,-66.293,-178.862,9.587,149.579
C02956=1133.099,223.239,-66.267,-178.865,9.583,149.579
C02957=1133.103,222.990,-66.242,-178.868,9.580,149.579
C02958=1133.108,222.741,-66.214,-178.871,9.577,149.579
C02959=1133.113,222.493,-66.189,-178.874,9.573,149.579
C02960=1133.117,222.244,-66.163,-178.877,9.570,149.579
C02961=1133.121,221.996,-66.137,-178.880,9.568,149.579
C02962=1133.126,221.747,-66.111,-178.883,9.564,149.579
C02963=1133.130,221.498,-66.085,-178.885,9.561,149.579
C02964=1133.134,221.250,-66.059,-178.888,9.557,149.579
C02965=1133.139,221.002,-66.033,-178.890,9.554,149.579
C02966=1133.144,220.753,-66.007,-178.894,9.551,149.579
C02967=1133.148,220.504,-65.981,-178.896,9.547,149.579
C02968=1133.152,220.255,-65.955,-178.899,9.544,149.579
C02969=1133.156,220.006,-65.929,-178.901,9.541,149.579
C02970=1133.162,219.759,-65.903,-178.904,9.538,149.578
C02971=1133.166,219.510,-65.877,-178.906,9.535,149.578
C02972=1133.170,219.261,-65.851,-178.909,9.532,149.578
C02973=1133.174,219.012,-65.825,-178.911,9.528,149.578
C02974=1133.178,218.763,-65.800,-178.913,9.525,149.578
C02975=1133.183,218.515,-65.774,-178.915,9.523,149.578
C02976=1133.188,218.266,-65.748,-178.918,9.520,149.578
C02977=1133.192,218.018,-65.721,-178.920,9.517,149.578
C02978=1133.196,217.769,-65.696,-178.922,9.513,149.578
C02979=1133.201,217.521,-65.670,-178.924,9.511,149.578
C02980=1133.205,217.272,-65.645,-178.927,9.508,149.578
C02981=1133.210,217.024,-65.619,-178.929,9.504,149.577
C02982=1133.214,216.775,-65.593,-178.931,9.502,149.577
C02983=1133.219,216.527,-65.568,-178.933,9.499,149.577
C02984=1133.223,216.278,-65.542,-178.935,9.496,149.577
C02985=1133.228,216.029,-65.516,-178.937,9.493,149.577
C02986=1133.233,215.781,-65.490,-178.939,9.490,149.577
C02987=1133.237,215.532,-65.464,-178.941,9.488,149.577
C02988=1133.241,215.283,-65.439,-178.943,9.485,149.576
C02989=1133.245,215.034,-65.413,-178.945,9.482,149.576
C02990=1133.250,214.786,-65.388,-178.946,9.480,149.576
C02991=1133.254,214.537,-65.362,-178.949,9.476,149.576
C02992=1133.259,214.288,-65.337,-178.950,9.474,149.576
C02993=1133.264,214.040,-65.311,-178.952,9.471,149.576
C02994=1133.268,213.791,-65.286,-178.954,9.469,149.575
C02995=1133.272,213.542,-65.260,-178.955,9.466,149.575
C02996=1133.277,213.294,-65.234,-178.957,9.464,149.575
C02997=1133.281,213.079,-65.212,-178.958,9.462,149.575
C02998=1133.284,212.865,-65.191,-178.960,9.459,149.575
C02999=1133.289,212.651,-65.168,-178.960,9.458,149.575
C03000=1133.292,212.436,-65.147,-178.961,9.456,149.574
C03001=1133.296,212.222,-65.125,-178.963,9.453,149.574
C03002=1133.300,212.008,-65.102,-178.964,9.451,149.574
C03003=1133.303,211.793,-65.081,-178.965,9.450,149.574
C03004=1133.308,211.579,-65.059,-178.967,9.447,149.574
C03005=1133.312,211.330,-65.033,-178.969,9.445,149.574
C03006=1133.317,211.082,-65.007,-178.970,9.442,149.574
C03007=1133.321,210.833,-64.982,-178.972,9.440,149.574
C03008=1133.325,210.584,-64.956,-178.974,9.437,149.574
C03009=1133.330,210.335,-64.931,-178.976,9.435,149.573
C03010=1133.335,210.087,-64.906,-178.978,9.433,149.573
C03011=1133.339,209.839,-64.881,-178.979,9.430,149.573
C03012=1133.343,209.590,-64.855,-178.981,9.428,149.573
C03013=1133.348,209.341,-64.830,-178.983,9.425,149.573
C03014=1133.352,209.093,-64.805,-178.985,9.423,149.573
C03015=1133.357,208.844,-64.779,-178.987,9.420,149.573
C03016=1133.361,208.596,-64.753,-178.990,9.418,149.573
C03017=1133.366,208.346,-64.728,-178.992,9.415,149.573
C03018=1133.370,208.097,-64.703,-178.994,9.413,149.573
C03019=1133.375,207.849,-64.677,-178.996,9.410,149.573
C03020=1133.380,207.600,-64.652,-178.999,9.407,149.573
C03021=1133.384,207.352,-64.627,-179.002,9.404,149.573
C03022=1133.388,207.103,-64.602,-179.003,9.402,149.573
C03023=1133.393,206.855,-64.577,-179.006,9.399,149.573
C03024=1133.397,206.606,-64.551,-179.009,9.396,149.573
C03025=1133.402,206.356,-64.526,-179.011,9.394,149.573
C03026=1133.407,206.108,-64.501,-179.014,9.391,149.573
C03027=1133.410,205.860,-64.476,-179.017,9.388,149.573
C03028=1133.415,205.611,-64.451,-179.020,9.386,149.574
C03029=1133.419,205.362,-64.425,-179.022,9.383,149.574
C03030=1133.425,205.113,-64.401,-179.025,9.380,149.574
C03031=1133.429,204.865,-64.375,-179.028,9.377,149.574
C03032=1133.433,204.616,-64.351,-179.031,9.374,149.574
C03033=1133.437,204.367,-64.325,-179.034,9.371,149.574
C03034=1133.443,204.119,-64.300,-179.037,9.368,149.574
C03035=1133.447,203.870,-64.275,-179.040,9.365,149.574
C03036=1133.451,203.621,-64.251,-179.043,9.362,149.574
C03037=1133.455,203.373,-64.225,-179.046,9.359,149.574
C03038=1133.460,203.124,-64.200,-179.050,9.356,149.575
C03039=1133.464,202.875,-64.176,-179.053,9.353,149.575
C03040=1133.469,202.627,-64.150,-179.056,9.350,149.575
C03041=1133.474,202.377,-64.125,-179.059,9.347,149.575
C03042=1133.478,202.129,-64.101,-179.063,9.343,149.575
C03043=1133.482,201.880,-64.075,-179.066,9.340,149.575
C03044=1133.487,201.631,-64.051,-179.069,9.337,149.575
C03045=1133.491,201.382,-64.026,-179.073,9.334,149.576
C03046=1133.496,201.134,-64.001,-179.076,9.330,149.576
C03047=1133.501,200.885,-63.976,-179.080,9.327,149.576
C03048=1133.505,200.636,-63.952,-179.084,9.323,149.576
C03049=1133.510,200.388,-63.926,-179.088,9.320,149.576
C03050=1133.514,200.139,-63.902,-179.091,9.317,149.577
C03051=1133.519,199.890,-63.877,-179.095,9.313,149.577
C03052=1133.523,199.642,-63.853,-179.098,9.309,149.577
C03053=1133.527,199.426,-63.832,-179.101,9.307,149.577
C03054=1133.531,199.212,-63.810,-179.105,9.303,149.577
C03055=1133.535,198.998,-63.789,-179.108,9.300,149.577
C03056=1133.539,198.783,-63.768,-179.111,9.297,149.577
C03057=1133.542,198.568,-63.746,-179.115,9.293,149.578
C03058=1133.546,198.354,-63.725,-179.119,9.290,149.578
C03059=1133.550,198.139,-63.705,-179.122,9.288,149.578
C03060=1133.555,197.924,-63.683,-179.126,9.284,149.578
C03061=1133.559,197.675,-63.659,-179.130,9.280,149.578
C03062=1133.564,197.426,-63.634,-179.133,9.276,149.578
C03063=1133.568,197.178,-63.610,-179.138,9.272,149.579
C03064=1133.572,196.929,-63.586,-179.142,9.268,149.579
C03065=1133.577,196.680,-63.561,-179.146,9.264,149.579
C03066=1133.581,196.432,-63.537,-179.151,9.259,149.579
C03067=1133.587,196.183,-63.512,-179.154,9.256,149.579
C03068=1133.590,195.934,-63.488,-179.156,9.253,149.579
C03069=1133.595,195.685,-63.464,-179.157,9.252,149.579
C03070=1133.600,195.437,-63.439,-179.158,9.249,149.579
C03071=1133.604,195.188,-63.415,-179.160,9.246,149.579
C03072=1133.608,194.939,-63.390,-179.161,9.244,149.578
C03073=1133.613,194.690,-63.366,-179.162,9.242,149.578
C03074=1133.618,194.442,-63.342,-179.164,9.239,149.578
C03075=1133.622,194.193,-63.318,-179.166,9.237,149.578
C03076=1133.627,193.944,-63.293,-179.167,9.234,149.578
C03077=1133.631,193.695,-63.269,-179.169,9.232,149.578
C03078=1133.636,193.447,-63.245,-179.170,9.229,149.577
C03079=1133.641,193.198,-63.220,-179.172,9.227,149.577
C03080=1133.645,192.949,-63.196,-179.174,9.224,149.577
C03081=1133.649,192.700,-63.173,-179.176,9.222,149.577
C03082=1133.654,192.451,-63.148,-179.177,9.219,149.577
C03083=1133.659,192.203,-63.124,-179.179,9.217,149.577
C03084=1133.663,191.954,-63.100,-179.181,9.214,149.577
C03085=1133.667,191.705,-63.076,-179.182,9.212,149.576
C03086=1133.672,191.456,-63.051,-179.185,9.208,149.576
C03087=1133.677,191.207,-63.027,-179.187,9.206,149.576
C03088=1133.681,190.959,-63.003,-179.188,9.203,149.576
C03089=1133.702,189.829,-62.895,-178.316,7.493,148.928
C03090=1133.706,189.580,-62.871,-178.318,7.490,148.928
C03091=1133.711,189.331,-62.847,-178.322,7.487,148.928
C03092=1133.716,189.082,-62.824,-178.324,7.485,148.928
C03093=1133.720,188.834,-62.800,-178.327,7.483,148.929
C03094=1133.725,188.585,-62.776,-178.330,7.480,148.929
C03095=1133.730,188.336,-62.753,-178.333,7.478,148.929
C03096=1133.734,188.087,-62.729,-178.336,7.475,148.929
C03097=1133.739,187.838,-62.706,-178.338,7.473,148.930
C03098=1133.743,187.589,-62.682,-178.341,7.470,148.930
C03099=1133.748,187.340,-62.659,-178.344,7.468,148.930
C03100=1133.752,187.092,-62.635,-178.347,7.466,148.930
C03101=1133.757,186.843,-62.611,-178.349,7.463,148.930
C03102=1133.762,186.594,-62.588,-178.353,7.460,148.931
C03103=1133.766,186.345,-62.565,-178.355,7.458,148.931
C03104=1133.770,186.097,-62.541,-178.358,7.456,148.931
C03105=1133.775,185.847,-62.518,-178.361,7.453,148.931
C03106=1133.780,185.598,-62.495,-178.364,7.451,148.932
C03107=1133.784,185.349,-62.471,-178.367,7.448,148.932
C03108=1133.790,185.101,-62.448,-178.370,7.446,148.932
C03109=1133.794,184.852,-62.425,-178.372,7.444,148.932
C03110=1133.799,184.603,-62.401,-178.375,7.441,148.932
C03111=1133.803,184.355,-62.378,-178.378,7.439,148.933
C03112=1133.807,184.106,-62.355,-178.381,7.437,148.933
C03113=1133.812,183.857,-62.331,-178.384,7.434,148.933
C03114=1133.817,183.587,-62.306,-178.387,7.431,148.933
C03115=1133.822,183.317,-62.281,-178.390,7.429,148.934
C03116=1133.827,183.047,-62.256,-178.393,7.427,148.934
C03117=1133.832,182.778,-62.231,-178.396,7.424,148.934
C03118=1133.836,182.529,-62.207,-178.399,7.421,148.935
C03119=1133.841,182.280,-62.184,-178.402,7.419,148.935
C03120=1133.846,182.031,-62.161,-178.405,7.417,148.935
C03121=1133.850,181.783,-62.138,-178.407,7.414,148.935
C03122=1133.855,181.534,-62.115,-178.410,7.412,148.936
C03123=1133.860,181.285,-62.091,-178.413,7.409,148.936
C03124=1133.864,181.036,-62.068,-178.416,7.407,148.936
C03125=1133.869,180.786,-62.046,-178.419,7.405,148.936
C03126=1133.873,180.537,-62.023,-178.422,7.402,148.937
C03127=1133.878,180.288,-61.999,-178.424,7.400,148.937
C03128=1133.883,180.040,-61.977,-178.427,7.398,148.937
C03129=1133.887,179.791,-61.954,-178.430,7.396,148.937
C03130=1133.892,179.542,-61.930,-178.433,7.393,148.938
C03131=1133.896,179.294,-61.907,-178.436,7.391,148.938
C03132=1133.901,179.045,-61.884,-178.438,7.388,148.938
C03133=1133.906,178.795,-61.861,-178.442,7.386,148.938
C03134=1133.910,178.547,-61.839,-178.444,7.384,148.939
C03135=1133.915,178.298,-61.816,-178.447,7.381,148.939
C03136=1133.920,178.049,-61.792,-178.450,7.378,148.939
C03137=1133.924,177.800,-61.770,-178.453,7.377,148.939
C03138=1133.929,177.551,-61.747,-178.456,7.374,148.940
C03139=1133.933,177.302,-61.725,-178.458,7.372,148.940
C03140=1133.938,177.053,-61.701,-178.462,7.370,148.940
C03141=1133.943,176.804,-61.679,-178.464,7.368,148.940
C03142=1133.947,176.555,-61.656,-178.467,7.365,148.941
C03143=1133.952,176.307,-61.633,-178.469,7.363,148.941
C03144=1133.956,176.058,-61.610,-178.473,7.360,148.941
C03145=1133.961,175.808,-61.587,-178.476,7.358,148.942
C03146=1133.965,175.560,-61.565,-178.478,7.356,148.942
C03147=1133.970,175.311,-61.542,-178.481,7.353,148.942
C03148=1133.975,175.062,-61.520,-178.484,7.351,148.942
C03149=1133.979,174.813,-61.496,-178.487,7.349,148.943
C03150=1133.985,174.564,-61.474,-178.490,7.347,148.943
C03151=1133.989,174.315,-61.451,-178.493,7.344,148.943
C03152=1133.994,174.066,-61.428,-178.495,7.342,148.943
C03153=1133.998,173.817,-61.406,-178.498,7.339,148.944
C03154=1134.003,173.569,-61.383,-178.501,7.338,148.944
C03155=1134.008,173.319,-61.361,-178.504,7.335,148.944
C03156=1134.012,173.070,-61.338,-178.506,7.333,148.944
C03157=1134.017,172.821,-61.316,-178.510,7.331,148.945
C03158=1134.021,172.573,-61.293,-178.512,7.328,148.945
C03159=1134.026,172.323,-61.270,-178.515,7.326,148.945
C03160=1134.031,172.075,-61.248,-178.518,7.324,148.946
C03161=1134.036,171.825,-61.225,-178.521,7.321,148.946
C03162=1134.040,171.577,-61.202,-178.524,7.319,148.946
C03163=1134.044,171.328,-61.181,-178.527,7.317,148.947
C03164=1134.049,171.079,-61.157,-178.529,7.314,148.947
C03165=1134.053,170.830,-61.135,-178.532,7.313,148.947
C03166=1134.059,170.581,-61.113,-178.535,7.310,148.947
C03167=1134.063,170.332,-61.090,-178.538,7.308,148.948
C03168=1134.068,170.083,-61.069,-178.541,7.306,148.948
C03169=1134.073,169.834,-61.046,-178.543,7.303,148.948
C03170=1134.077,169.585,-61.023,-178.547,7.301,148.948
C03171=1134.082,169.336,-61.002,-178.549,7.299,148.949
C03172=1134.086,169.087,-60.978,-178.552,7.296,148.949
C03173=1134.091,168.839,-60.957,-178.555,7.295,148.949
C03174=1134.096,168.589,-60.934,-178.558,7.292,148.950
C03175=1134.101,168.340,-60.912,-178.560,7.290,148.950
C03176=1134.105,168.092,-60.889,-178.564,7.288,148.950
C03177=1134.109,167.842,-60.867,-178.566,7.286,148.950
C03178=1134.115,167.593,-60.845,-178.569,7.283,148.951
C03179=1134.119,167.344,-60.823,-178.572,7.281,148.951
C03180=1134.124,167.096,-60.801,-178.575,7.279,148.951
C03181=1134.128,166.847,-60.779,-178.577,7.277,148.952
C03182=1134.134,166.598,-60.756,-178.581,7.274,148.952
C03183=1134.138,166.348,-60.734,-178.583,7.272,148.952
C03184=1134.142,166.099,-60.712,-178.586,7.270,148.952
C03185=1134.147,165.851,-60.690,-178.589,7.268,148.953
C03186=1134.152,165.601,-60.667,-178.592,7.266,148.953
C03187=1134.157,165.353,-60.645,-178.595,7.263,148.953
C03188=1134.161,165.103,-60.623,-178.597,7.261,148.954
C03189=1134.166,164.855,-60.602,-178.601,7.259,148.954
C03190=1134.170,164.605,-60.580,-178.603,7.257,148.954
C03191=1134.175,164.357,-60.558,-178.606,7.254,148.955
C03192=1134.180,164.108,-60.535,-178.609,7.253,148.955
C03193=1134.185,163.859,-60.513,-178.612,7.250,148.955
C03194=1134.189,163.610,-60.491,-178.614,7.248,148.955
C03195=1134.194,163.361,-60.469,-178.618,7.246,148.956
C03196=1134.198,163.112,-60.447,-178.620,7.244,148.956
C03197=1134.203,162.863,-60.426,-178.623,7.242,148.956
C03198=1134.207,162.614,-60.403,-178.626,7.239,148.957
C03199=1134.212,162.365,-60.382,-178.629,7.238,148.957
C03200=1134.218,162.116,-60.360,-178.631,7.235,148.957
C03201=1134.222,161.867,-60.337,-178.634,7.233,148.958
C03202=1134.227,161.618,-60.316,-178.637,7.230,148.958
C03203=1134.231,161.369,-60.294,-178.640,7.228,148.958
C03204=1134.236,161.120,-60.272,-178.643,7.226,148.958
C03205=1134.240,160.871,-60.250,-178.646,7.224,148.959
C03206=1134.245,160.622,-60.229,-178.648,7.222,148.959
C03207=1134.250,160.372,-60.207,-178.651,7.220,148.959
C03208=1134.254,160.124,-60.185,-178.654,7.218,148.960
C03209=1134.259,159.875,-60.164,-178.657,7.215,148.960
C03210=1134.264,159.626,-60.142,-178.659,7.213,148.960
C03211=1134.268,159.377,-60.120,-178.663,7.211,148.961
C03212=1134.273,159.128,-60.098,-178.665,7.209,148.961
C03213=1134.278,158.878,-60.077,-178.668,7.207,148.961
C03214=1134.283,158.630,-60.055,-178.671,7.204,148.961
C03215=1134.287,158.380,-60.033,-178.674,7.203,148.962
C03216=1134.292,158.132,-60.011,-178.677,7.200,148.962
C03217=1134.297,157.883,-59.990,-178.680,7.199,148.963
C03218=1134.302,157.614,-59.966,-178.683,7.196,148.963
C03219=1134.307,157.345,-59.944,-178.685,7.194,148.963
C03220=1134.312,157.076,-59.920,-178.689,7.191,148.963
C03221=1134.317,156.807,-59.897,-178.692,7.189,148.964
C03222=1134.321,156.558,-59.875,-178.695,7.187,148.964
C03223=1134.326,156.308,-59.854,-178.697,7.186,148.965
C03224=1134.331,156.060,-59.832,-178.700,7.183,148.965
C03225=1134.335,155.810,-59.810,-178.703,7.181,148.965
C03226=1134.340,155.562,-59.788,-178.706,7.178,148.966
C03227=1134.346,155.313,-59.767,-178.709,7.177,148.966
C03228=1134.350,155.064,-59.746,-178.711,7.175,148.966
C03229=1134.354,154.814,-59.725,-178.714,7.172,148.966
C03230=1134.359,154.566,-59.703,-178.717,7.170,148.967
C03231=1134.364,154.317,-59.682,-178.720,7.168,148.967
C03232=1134.369,154.067,-59.660,-178.723,7.166,148.967
C03233=1134.373,153.818,-59.639,-178.725,7.164,148.968
C03234=1134.378,153.569,-59.618,-178.729,7.162,148.968
C03235=1134.383,153.321,-59.597,-178.731,7.160,148.968
C03236=1134.387,153.071,-59.575,-178.734,7.158,148.969
C03237=1134.392,152.822,-59.554,-178.737,7.155,148.969
C03238=1134.397,152.574,-59.532,-178.740,7.154,148.969
C03239=1134.401,152.325,-59.512,-178.742,7.152,148.970
C03240=1134.406,152.075,-59.489,-178.746,7.149,148.970
C03241=1134.411,151.826,-59.469,-178.748,7.147,148.970
C03242=1134.416,151.577,-59.447,-178.751,7.145,148.971
C03243=1134.420,151.328,-59.426,-178.754,7.143,148.971
C03244=1134.425,151.078,-59.405,-178.757,7.142,148.971
C03245=1134.430,150.830,-59.383,-178.760,7.139,148.972
C03246=1134.435,150.581,-59.362,-178.762,7.137,148.972
C03247=1134.439,150.332,-59.341,-178.765,7.135,148.972
C03248=1134.444,150.083,-59.320,-178.768,7.133,148.973
C03249=1134.449,149.833,-59.299,-178.771,7.131,148.973
C03250=1134.454,149.584,-59.277,-178.774,7.129,148.973
C03251=1134.458,149.335,-59.257,-178.777,7.126,148.974
C03252=1134.463,149.087,-59.235,-178.779,7.125,148.974
C03253=1134.468,148.837,-59.214,-178.782,7.123,148.974
C03254=1134.472,148.589,-59.194,-178.785,7.121,148.975
C03255=1134.477,148.339,-59.172,-178.788,7.119,148.975
C03256=1134.482,148.090,-59.151,-178.791,7.117,148.976
C03257=1134.486,147.841,-59.131,-178.794,7.114,148.976
C03258=1134.492,147.592,-59.110,-178.796,7.113,148.976
C03259=1134.496,147.343,-59.089,-178.799,7.111,148.976
C03260=1134.501,147.094,-59.068,-178.802,7.108,148.977
C03261=1134.506,146.845,-59.047,-178.805,7.107,148.977
C03262=1134.510,146.595,-59.026,-178.807,7.105,148.977
C03263=1134.515,146.347,-59.004,-178.811,7.102,148.978
C03264=1134.519,146.098,-58.984,-178.813,7.100,148.978
C03265=1134.524,145.848,-58.963,-178.816,7.099,148.979
C03266=1134.529,145.599,-58.942,-178.819,7.097,148.979
C03267=1134.534,145.350,-58.922,-178.822,7.094,148.979
C03268=1134.539,145.102,-58.900,-178.824,7.092,148.979
C03269=1134.543,144.853,-58.879,-178.827,7.091,148.980
C03270=1134.548,144.603,-58.859,-178.830,7.088,148.980
C03271=1134.553,144.354,-58.838,-178.833,7.087,148.981
C03272=1134.557,144.104,-58.817,-178.836,7.085,148.981
C03273=1134.562,143.855,-58.796,-178.839,7.082,148.981
C03274=1134.567,143.606,-58.775,-178.842,7.081,148.982
C03275=1134.572,143.357,-58.755,-178.844,7.079,148.982
C03276=1134.577,143.108,-58.734,-178.847,7.077,148.982
C03277=1134.581,142.860,-58.713,-178.850,7.074,148.983
C03278=1134.586,142.610,-58.692,-178.853,7.073,148.983
C03279=1134.590,142.361,-58.672,-178.856,7.071,148.983
C03280=1134.595,142.113,-58.651,-178.859,7.068,148.984
C03281=1134.600,141.863,-58.630,-178.862,7.067,148.984
C03282=1134.604,141.614,-58.610,-178.864,7.065,148.984
C03283=1134.610,141.365,-58.589,-178.867,7.063,148.985
C03284=1134.614,141.116,-58.569,-178.870,7.060,148.985
C03285=1134.619,140.867,-58.548,-178.873,7.059,148.986
C03286=1134.624,140.618,-58.527,-178.875,7.057,148.986
C03287=1134.628,140.368,-58.508,-178.878,7.055,148.986
C03288=1134.634,140.119,-58.487,-178.881,7.053,148.987
C03289=1134.638,139.870,-58.466,-178.884,7.051,148.987
C03290=1134.642,139.621,-58.446,-178.886,7.049,148.987
C03291=1134.648,139.372,-58.425,-178.889,7.047,148.988
C03292=1134.652,139.123,-58.405,-178.892,7.045,148.988
C03293=1134.657,138.874,-58.384,-178.895,7.043,148.988
C03294=1134.662,138.625,-58.363,-178.898,7.042,148.989
C03295=1134.666,138.376,-58.343,-178.900,7.040,148.989
C03296=1134.671,138.126,-58.323,-178.904,7.037,148.990
C03297=1134.676,137.877,-58.302,-178.906,7.036,148.990
C03298=1134.681,137.628,-58.282,-178.909,7.034,148.990
C03299=1134.685,137.379,-58.262,-178.911,7.032,148.991
C03300=1134.690,137.130,-58.241,-178.915,7.029,148.991
C03301=1134.695,136.880,-58.221,-178.918,7.028,148.991
C03302=1134.699,136.631,-58.201,-178.920,7.026,148.992
C03303=1134.704,136.383,-58.181,-178.923,7.024,148.992
C03304=1134.710,136.134,-58.160,-178.926,7.022,148.993
C03305=1134.714,135.884,-58.140,-178.929,7.020,148.993
C03306=1134.719,135.635,-58.120,-178.932,7.018,148.993
C03307=1134.723,135.386,-58.099,-178.934,7.017,148.994
C03308=1134.729,135.136,-58.079,-178.937,7.014,148.994
C03309=1134.733,134.887,-58.059,-178.940,7.012,148.994
C03310=1134.737,134.639,-58.038,-178.943,7.011,148.995
C03311=1134.742,134.389,-58.019,-178.945,7.009,148.995
C03312=1134.747,134.141,-57.999,-178.948,7.007,148.995
C03313=1134.752,133.891,-57.978,-178.951,7.005,148.996
C03314=1134.757,133.642,-57.958,-178.954,7.003,148.996
C03315=1134.762,133.393,-57.938,-178.957,7.001,148.997
C03316=1134.766,133.144,-57.917,-178.960,7.000,148.997
C03317=1134.771,132.894,-57.897,-178.962,6.998,148.997
C03318=1134.776,132.645,-57.877,-178.966,6.995,148.998
C03319=1134.781,132.396,-57.857,-178.968,6.994,148.998
C03320=1134.786,132.147,-57.837,-178.971,6.992,148.998
C03321=1134.790,131.898,-57.817,-178.973,6.990,148.999
C03322=1134.795,131.630,-57.795,-178.977,6.988,148.999
C03323=1134.801,131.361,-57.774,-178.980,6.986,149.000
C03324=1134.806,131.092,-57.753,-178.983,6.984,149.000
C03325=1134.811,130.824,-57.730,-178.986,6.982,149.001
C03326=1134.816,130.574,-57.711,-178.989,6.980,149.001
C03327=1134.820,130.325,-57.690,-178.991,6.979,149.001
C03328=1134.826,130.076,-57.671,-178.995,6.976,149.002
C03329=1134.830,129.827,-57.651,-178.997,6.974,149.002
C03330=1134.835,129.578,-57.631,-179.000,6.972,149.002
C03331=1134.839,129.328,-57.611,-179.002,6.971,149.003
C03332=1134.845,129.080,-57.591,-179.005,6.969,149.003
C03333=1134.849,128.831,-57.572,-179.008,6.967,149.003
C03334=1134.854,128.582,-57.551,-179.011,6.965,149.004
C03335=1134.858,128.332,-57.532,-179.014,6.963,149.004
C03336=1134.864,128.083,-57.512,-179.017,6.961,149.005
C03337=1134.868,127.834,-57.492,-179.019,6.960,149.005
C03338=1134.873,127.585,-57.472,-179.022,6.958,149.005
C03339=1134.878,127.335,-57.453,-179.025,6.956,149.006
C03340=1134.883,127.087,-57.433,-179.028,6.954,149.006
C03341=1134.887,126.837,-57.413,-179.031,6.952,149.007
C03342=1134.892,126.588,-57.393,-179.034,6.950,149.007
C03343=1134.897,126.339,-57.373,-179.036,6.949,149.007
C03344=1134.902,126.090,-57.354,-179.039,6.947,149.008
C03345=1134.907,125.840,-57.334,-179.042,6.945,149.008
C03346=1134.911,125.591,-57.314,-179.044,6.944,149.009
C03347=1134.917,125.342,-57.294,-179.048,6.941,149.009
C03348=1134.921,125.093,-57.275,-179.051,6.940,149.009
C03349=1134.925,124.844,-57.256,-179.053,6.938,149.010
C03350=1134.931,124.595,-57.236,-179.056,6.936,149.010
C03351=1134.935,124.345,-57.217,-179.059,6.934,149.011
C03352=1134.940,124.096,-57.196,-179.061,6.933,149.011
C03353=1134.945,123.847,-57.177,-179.064,6.931,149.011
C03354=1134.950,123.598,-57.157,-179.067,6.929,149.012
C03355=1134.955,123.348,-57.138,-179.070,6.927,149.012
C03356=1134.960,123.099,-57.118,-179.073,6.925,149.013
C03357=1134.964,122.850,-57.099,-179.076,6.924,149.013
C03358=1134.969,122.601,-57.080,-179.078,6.922,149.013
C03359=1134.974,122.352,-57.060,-179.081,6.920,149.014
C03360=1134.978,122.103,-57.040,-179.084,6.918,149.014
C03361=1134.983,121.853,-57.020,-179.087,6.917,149.015
C03362=1134.988,121.605,-57.002,-179.089,6.915,149.015
C03363=1134.993,121.355,-56.982,-179.093,6.913,149.015
C03364=1134.998,121.106,-56.963,-179.095,6.911,149.016
C03365=1135.003,120.857,-56.943,-179.098,6.909,149.016
C03366=1135.007,120.607,-56.923,-179.101,6.908,149.017
C03367=1135.012,120.358,-56.905,-179.104,6.906,149.017
C03368=1135.017,120.109,-56.885,-179.106,6.904,149.017
C03369=1135.022,119.860,-56.866,-179.109,6.903,149.018
C03370=1135.027,119.610,-56.846,-179.112,6.901,149.018
C03371=1135.031,119.362,-56.827,-179.114,6.899,149.019
C03372=1135.036,119.112,-56.808,-179.118,6.897,149.019
C03373=1135.041,118.863,-56.788,-179.121,6.895,149.019
C03374=1135.046,118.614,-56.769,-179.123,6.893,149.020
C03375=1135.050,118.365,-56.750,-179.126,6.892,149.020
C03376=1135.056,118.116,-56.730,-179.129,6.890,149.021
C03377=1135.061,117.866,-56.711,-179.131,6.888,149.021
C03378=1135.065,117.617,-56.693,-179.134,6.887,149.021
C03379=1135.070,117.367,-56.673,-179.137,6.885,149.022
C03380=1135.075,117.119,-56.654,-179.140,6.883,149.022
C03381=1135.079,116.869,-56.635,-179.142,6.882,149.023
C03382=1135.085,116.621,-56.615,-179.145,6.880,149.023
C03383=1135.089,116.371,-56.596,-179.148,6.878,149.024
C03384=1135.094,116.122,-56.578,-179.151,6.876,149.024
C03385=1135.099,115.872,-56.558,-179.154,6.874,149.024
C03386=1135.104,115.624,-56.539,-179.157,6.872,149.025
C03387=1135.108,115.374,-56.520,-179.159,6.871,149.025
C03388=1135.114,115.125,-56.501,-179.162,6.869,149.026
C03389=1135.118,114.875,-56.482,-179.165,6.867,149.026
C03390=1135.123,114.626,-56.463,-179.168,6.866,149.026
C03391=1135.127,114.377,-56.444,-179.170,6.864,149.027
C03392=1135.133,114.128,-56.425,-179.173,6.862,149.027
C03393=1135.138,113.878,-56.406,-179.176,6.861,149.028
C03394=1135.142,113.630,-56.387,-179.178,6.859,149.028
C03395=1135.147,113.380,-56.367,-179.181,6.857,149.028
C03396=1135.152,113.131,-56.349,-179.184,6.856,149.029
C03397=1135.157,112.881,-56.330,-179.187,6.854,149.029
C03398=1135.161,112.633,-56.311,-179.189,6.852,149.030
C03399=1135.167,112.383,-56.292,-179.193,6.851,149.030
C03400=1135.171,112.134,-56.273,-179.195,6.849,149.031
C03401=1135.176,111.885,-56.254,-179.198,6.847,149.031
C03402=1135.181,111.635,-56.236,-179.201,6.846,149.031
C03403=1135.186,111.386,-56.216,-179.204,6.844,149.032
C03404=1135.191,111.137,-56.198,-179.206,6.842,149.032
C03405=1135.196,110.888,-56.179,-179.209,6.841,149.033
C03406=1135.200,110.639,-56.160,-179.212,6.838,149.033
C03407=1135.205,110.389,-56.141,-179.215,6.837,149.033
C03408=1135.210,110.140,-56.122,-179.218,6.835,149.034
C03409=1135.216,109.891,-56.104,-179.221,6.833,149.034
C03410=1135.220,109.642,-56.085,-179.223,6.832,149.035
C03411=1135.225,109.392,-56.067,-179.226,6.830,149.035
C03412=1135.229,109.143,-56.047,-179.229,6.828,149.036
C03413=1135.234,108.894,-56.029,-179.231,6.827,149.036
C03414=1135.240,108.645,-56.010,-179.234,6.825,149.036
C03415=1135.244,108.395,-55.991,-179.237,6.824,149.037
C03416=1135.249,108.146,-55.973,-179.240,6.822,149.037
C03417=1135.254,107.897,-55.954,-179.243,6.820,149.038
C03418=1135.258,107.648,-55.935,-179.246,6.819,149.038
C03419=1135.264,107.398,-55.917,-179.248,6.817,149.039
C03420=1135.269,107.149,-55.899,-179.251,6.815,149.039
C03421=1135.273,106.900,-55.880,-179.254,6.814,149.039
C03422=1135.278,106.650,-55.861,-179.257,6.812,149.040
C03423=1135.283,106.402,-55.842,-179.259,6.810,149.040
C03424=1135.287,106.152,-55.824,-179.262,6.809,149.041
C03425=1135.293,105.902,-55.805,-179.265,6.807,149.041
C03426=1135.298,105.635,-55.785,-179.268,6.806,149.042
C03427=1135.304,105.366,-55.765,-179.271,6.804,149.042
C03428=1135.309,105.098,-55.746,-179.273,6.802,149.043
C03429=1135.313,104.829,-55.726,-179.277,6.800,149.043
C03430=1135.318,104.580,-55.707,-179.279,6.799,149.043
C03431=1135.323,104.331,-55.689,-179.282,6.798,149.044
C03432=1135.328,104.082,-55.671,-179.285,6.796,149.044
C03433=1135.333,103.831,-55.652,-179.288,6.794,149.045
C03434=1135.338,103.583,-55.633,-179.290,6.793,149.045
C03435=1135.343,103.334,-55.615,-179.293,6.791,149.046
C03436=1135.348,103.085,-55.597,-179.296,6.789,149.046
C03437=1135.353,102.834,-55.578,-179.299,6.787,149.047
C03438=1135.357,102.586,-55.560,-179.301,6.786,149.047
C03439=1135.362,102.337,-55.542,-179.304,6.784,149.047
C03440=1135.367,102.087,-55.524,-179.307,6.782,149.048
C03441=1135.372,101.838,-55.505,-179.310,6.781,149.048
C03442=1135.377,101.588,-55.487,-179.313,6.780,149.049
C03443=1135.382,101.339,-55.469,-179.315,6.778,149.049
C03444=1135.387,101.090,-55.450,-179.318,6.776,149.050
C03445=1135.392,100.841,-55.432,-179.321,6.774,149.050
C03446=1135.396,100.591,-55.414,-179.324,6.773,149.050
C03447=1135.401,100.342,-55.396,-179.326,6.771,149.051
C03448=1135.407,100.093,-55.377,-179.329,6.769,149.051
C03449=1135.411,99.843,-55.359,-179.332,6.768,149.052
C03450=1135.416,99.594,-55.341,-179.335,6.767,149.052
C03451=1135.421,99.344,-55.323,-179.338,6.765,149.053
C03452=1135.426,99.095,-55.305,-179.341,6.763,149.053
C03453=1135.430,98.847,-55.286,-179.343,6.762,149.054
C03454=1135.435,98.598,-55.268,-179.345,6.761,149.054
C03455=1135.440,98.348,-55.250,-179.348,6.759,149.054
C03456=1135.445,98.099,-55.232,-179.351,6.757,149.055
C03457=1135.450,97.849,-55.213,-179.354,6.756,149.055
C03458=1135.455,97.600,-55.195,-179.357,6.754,149.056
C03459=1135.460,97.351,-55.177,-179.360,6.753,149.056
C03460=1135.465,97.101,-55.159,-179.362,6.751,149.057
C03461=1135.470,96.852,-55.141,-179.365,6.749,149.057
C03462=1135.475,96.602,-55.124,-179.368,6.748,149.058
C03463=1135.480,96.353,-55.106,-179.371,6.746,149.058
C03464=1135.485,96.104,-55.088,-179.373,6.744,149.058
C03465=1135.489,95.854,-55.070,-179.376,6.743,149.059
C03466=1135.494,95.605,-55.052,-179.379,6.742,149.059
C03467=1135.499,95.356,-55.034,-179.381,6.740,149.060
C03468=1135.504,95.107,-55.016,-179.384,6.739,149.060
C03469=1135.509,94.858,-54.998,-179.387,6.737,149.061
C03470=1135.514,94.608,-54.980,-179.390,6.735,149.061
C03471=1135.518,94.359,-54.962,-179.392,6.734,149.062
C03472=1135.524,94.109,-54.945,-179.396,6.733,149.062
C03473=1135.529,93.860,-54.927,-179.398,6.731,149.063
C03474=1135.533,93.611,-54.909,-179.401,6.729,149.063
C03475=1135.538,93.362,-54.891,-179.404,6.728,149.063
C03476=1135.543,93.113,-54.873,-179.406,6.727,149.064
C03477=1135.548,92.864,-54.855,-179.409,6.725,149.064
C03478=1135.553,92.613,-54.837,-179.411,6.723,149.065
C03479=1135.557,92.364,-54.820,-179.415,6.722,149.065
C03480=1135.562,92.115,-54.802,-179.417,6.720,149.066
C03481=1135.567,91.866,-54.784,-179.420,6.719,149.066
C03482=1135.572,91.616,-54.766,-179.423,6.717,149.067
C03483=1135.577,91.367,-54.749,-179.426,6.715,149.067
C03484=1135.582,91.118,-54.731,-179.428,6.715,149.068
C03485=1135.587,90.868,-54.713,-179.431,6.713,149.068
C03486=1135.592,90.619,-54.695,-179.434,6.712,149.069
C03487=1135.596,90.370,-54.678,-179.436,6.710,149.069
C03488=1135.601,90.121,-54.660,-179.439,6.708,149.069
C03489=1135.606,89.871,-54.643,-179.442,6.707,149.070
C03490=1135.611,89.622,-54.625,-179.445,6.705,149.070
C03491=1135.616,89.373,-54.607,-179.448,6.704,149.071
C03492=1135.621,89.123,-54.589,-179.450,6.703,149.071
C03493=1135.626,88.874,-54.572,-179.453,6.701,149.072
C03494=1135.631,88.624,-54.555,-179.456,6.699,149.072
C03495=1135.636,88.375,-54.537,-179.458,6.698,149.073
C03496=1135.641,88.126,-54.519,-179.461,6.696,149.073
C03497=1135.646,87.877,-54.502,-179.464,6.695,149.074
C03498=1135.651,87.628,-54.485,-179.467,6.693,149.074
C03499=1135.656,87.378,-54.467,-179.469,6.692,149.075
C03500=1135.661,87.129,-54.449,-179.472,6.691,149.075
C03501=1135.666,86.879,-54.432,-179.475,6.689,149.075
C03502=1135.670,86.630,-54.415,-179.477,6.687,149.076
C03503=1135.675,86.380,-54.397,-179.481,6.686,149.076
C03504=1135.680,86.131,-54.379,-179.483,6.684,149.077
C03505=1135.685,85.881,-54.362,-179.485,6.684,149.077
C03506=1135.690,85.632,-54.345,-179.488,6.682,149.078
C03507=1135.695,85.383,-54.327,-179.491,6.680,149.078
C03508=1135.700,85.134,-54.310,-179.494,6.679,149.079
C03509=1135.705,84.884,-54.292,-179.497,6.677,149.079
C03510=1135.710,84.636,-54.275,-179.500,6.676,149.080
C03511=1135.715,84.386,-54.258,-179.502,6.675,149.080
C03512=1135.720,84.137,-54.240,-179.505,6.673,149.080
C03513=1135.724,83.887,-54.223,-179.507,6.671,149.081
C03514=1135.730,83.637,-54.206,-179.511,6.670,149.082
C03515=1135.734,83.388,-54.188,-179.513,6.668,149.082
C03516=1135.739,83.139,-54.171,-179.515,6.668,149.082
C03517=1135.744,82.889,-54.153,-179.518,6.666,149.083
C03518=1135.749,82.641,-54.137,-179.521,6.664,149.083
C03519=1135.754,82.391,-54.120,-179.524,6.663,149.084
C03520=1135.759,82.142,-54.102,-179.527,6.661,149.084
C03521=1135.764,81.892,-54.085,-179.529,6.660,149.085
C03522=1135.769,81.642,-54.068,-179.532,6.659,149.085
C03523=1135.773,81.394,-54.051,-179.535,6.657,149.086
C03524=1135.779,81.144,-54.034,-179.538,6.656,149.086
C03525=1135.784,80.895,-54.016,-179.540,6.654,149.087
C03526=1135.788,80.645,-54.000,-179.543,6.653,149.087
C03527=1135.793,80.396,-53.982,-179.545,6.652,149.088
C03528=1135.798,80.147,-53.965,-179.548,6.650,149.088
C03529=1135.804,79.897,-53.948,-179.551,6.649,149.089
C03530=1135.809,79.629,-53.929,-179.554,6.647,149.089
C03531=1135.814,79.360,-53.911,-179.557,6.645,149.090
C03532=1135.820,79.092,-53.893,-179.560,6.644,149.090
C03533=1135.824,78.823,-53.875,-179.563,6.643,149.091
C03534=1135.829,78.574,-53.857,-179.566,6.641,149.091
C03535=1135.834,78.325,-53.841,-179.568,6.640,149.092
C03536=1135.840,78.076,-53.823,-179.571,6.639,149.092
C03537=1135.844,77.826,-53.807,-179.574,6.637,149.093
C03538=1135.849,77.576,-53.789,-179.576,6.635,149.093
C03539=1135.854,77.327,-53.773,-179.579,6.635,149.093
C03540=1135.859,77.078,-53.755,-179.582,6.633,149.094
C03541=1135.864,76.829,-53.739,-179.585,6.632,149.094
C03542=1135.869,76.579,-53.721,-179.587,6.630,149.095
C03543=1135.874,76.330,-53.705,-179.590,6.628,149.095
C03544=1135.879,76.080,-53.688,-179.593,6.628,149.096
C03545=1135.884,75.831,-53.671,-179.595,6.626,149.096
C03546=1135.889,75.581,-53.654,-179.598,6.625,149.097
C03547=1135.894,75.332,-53.637,-179.601,6.623,149.097
C03548=1135.899,75.083,-53.621,-179.603,6.622,149.098
C03549=1135.904,74.833,-53.604,-179.606,6.621,149.098
C03550=1135.909,74.584,-53.587,-179.609,6.619,149.099
C03551=1135.914,74.335,-53.570,-179.612,6.617,149.099
C03552=1135.919,74.085,-53.553,-179.614,6.617,149.100
C03553=1135.924,73.836,-53.537,-179.617,6.615,149.100
C03554=1135.929,73.586,-53.520,-179.620,6.614,149.101
C03555=1135.933,73.337,-53.503,-179.623,6.612,149.101
C03556=1135.938,73.087,-53.486,-179.625,6.611,149.102
C03557=1135.944,72.838,-53.469,-179.628,6.610,149.102
C03558=1135.948,72.589,-53.453,-179.631,6.608,149.103
C03559=1135.953,72.339,-53.436,-179.633,6.607,149.103
C03560=1135.958,72.090,-53.419,-179.636,6.606,149.104
C03561=1135.963,71.841,-53.403,-179.638,6.604,149.104
C03562=1135.968,71.592,-53.386,-179.642,6.603,149.105
C03563=1135.973,71.342,-53.369,-179.644,6.602,149.105
C03564=1135.978,71.093,-53.352,-179.647,6.600,149.106
C03565=1135.983,70.843,-53.337,-179.649,6.599,149.106
C03566=1135.988,70.594,-53.319,-179.653,6.597,149.107
C03567=1135.993,70.344,-53.303,-179.655,6.597,149.107
C03568=1135.998,70.095,-53.287,-179.657,6.595,149.107
C03569=1136.002,69.846,-53.270,-179.660,6.593,149.108
C03570=1136.008,69.597,-53.253,-179.663,6.593,149.109
C03571=1136.013,69.347,-53.237,-179.666,6.591,149.109
C03572=1136.017,69.097,-53.220,-179.668,6.589,149.109
C03573=1136.022,68.848,-53.204,-179.671,6.589,149.110
C03574=1136.028,68.599,-53.187,-179.674,6.587,149.111
C03575=1136.033,68.350,-53.170,-179.676,6.586,149.111
C03576=1136.038,68.100,-53.155,-179.679,6.584,149.111
C03577=1136.042,67.850,-53.138,-179.681,6.583,149.112
C03578=1136.047,67.601,-53.122,-179.685,6.582,149.112
C03579=1136.052,67.352,-53.104,-179.687,6.580,149.113
C03580=1136.058,67.102,-53.089,-179.690,6.579,149.113
C03581=1136.062,66.853,-53.072,-179.692,6.578,149.114
C03582=1136.067,66.604,-53.056,-179.696,6.577,149.114
C03583=1136.072,66.354,-53.040,-179.698,6.576,149.115
C03584=1136.078,66.105,-53.023,-179.700,6.574,149.115
C03585=1136.082,65.855,-53.006,-179.703,6.572,149.116
C03586=1136.087,65.605,-52.990,-179.706,6.572,149.116
C03587=1136.092,65.356,-52.974,-179.709,6.570,149.117
C03588=1136.097,65.107,-52.957,-179.711,6.569,149.117
C03589=1136.102,64.857,-52.942,-179.714,6.567,149.118
C03590=1136.107,64.608,-52.925,-179.717,6.566,149.118
C03591=1136.112,64.359,-52.909,-179.719,6.565,149.119
C03592=1136.117,64.109,-52.892,-179.722,6.563,149.119
C03593=1136.122,63.860,-52.876,-179.725,6.563,149.120
C03594=1136.127,63.610,-52.860,-179.728,6.561,149.120
C03595=1136.132,63.361,-52.844,-179.730,6.559,149.121
C03596=1136.137,63.111,-52.828,-179.733,6.559,149.121
C03597=1136.142,62.862,-52.811,-179.736,6.557,149.122
C03598=1136.147,62.612,-52.795,-179.738,6.556,149.122
C03599=1136.152,62.363,-52.779,-179.741,6.555,149.123
C03600=1136.157,62.113,-52.763,-179.743,6.553,149.123
C03601=1136.162,61.864,-52.747,-179.746,6.553,149.124
C03602=1136.166,61.614,-52.731,-179.749,6.551,149.124
C03603=1136.172,61.366,-52.715,-179.752,6.549,149.125
C03604=1136.177,61.116,-52.699,-179.754,6.549,149.125
C03605=1136.181,60.867,-52.682,-179.757,6.547,149.126
C03606=1136.187,60.617,-52.667,-179.760,6.546,149.126
C03607=1136.191,60.368,-52.650,-179.762,6.545,149.127
C03608=1136.197,60.118,-52.634,-179.765,6.544,149.127
C03609=1136.201,59.869,-52.618,-179.768,6.542,149.128
C03610=1136.207,59.620,-52.602,-179.770,6.541,149.128
C03611=1136.212,59.370,-52.587,-179.773,6.539,149.129
C03612=1136.216,59.121,-52.570,-179.776,6.538,149.129
C03613=1136.222,58.871,-52.554,-179.778,6.537,149.130
C03614=1136.226,58.622,-52.538,-179.781,6.536,149.130
C03615=1136.232,58.372,-52.522,-179.784,6.535,149.131
C03616=1136.237,58.123,-52.507,-179.786,6.534,149.131
C03617=1136.242,57.873,-52.490,-179.789,6.532,149.132
C03618=1136.247,57.624,-52.474,-179.791,6.531,149.132
C03619=1136.252,57.374,-52.458,-179.794,6.530,149.133
C03620=1136.257,57.125,-52.442,-179.797,6.528,149.133
C03621=1136.262,56.876,-52.426,-179.799,6.527,149.134
C03622=1136.266,56.626,-52.411,-179.803,6.526,149.134
C03623=1136.271,56.377,-52.395,-179.805,6.525,149.135
C03624=1136.277,56.128,-52.379,-179.808,6.524,149.135
C03625=1136.281,55.878,-52.363,-179.810,6.522,149.136
